LIN {X 0,Y 136.185,Z 195.521,A -85,B 0,C 180,E1 -24638.251,E2 -24638.251} C_VEL
LIN {X 0,Y 136.232,Z 195.509,A -85,B 0,C 180,E1 -24641.969,E2 -24641.969} C_VEL
LIN {X 0,Y 136.486,Z 195.483,A -85,B 0,C 180,E1 -24648.113,E2 -24648.113} C_VEL
LIN {X 0,Y 136.58,Z 195.466,A -85,B 0,C 180,E1 -24651.119,E2 -24651.119} C_VEL
LIN {X 0,Y 137.121,Z 195.397,A -85,B 0,C 180,E1 -24660,E2 -24660} C_VEL
LIN {X 0,Y 136.58,Z 195.467,A -85,B 0,C 180,E1 -24668.88,E2 -24668.88} C_VEL
LIN {X 0,Y 136.479,Z 195.483,A -85,B 0,C 180,E1 -24671.955,E2 -24671.955} C_VEL
LIN {X 0,Y 136.232,Z 195.509,A -85,B 0,C 180,E1 -24678.031,E2 -24678.031} C_VEL
LIN {X 0,Y 136.184,Z 195.521,A -85,B 0,C 180,E1 -24681.747,E2 -24681.747} C_VEL
LIN {X 0,Y 136.081,Z 195.533,A -85,B 0,C 180,E1 -24688.612,E2 -24688.612} C_VEL
LIN {X 0,Y 136.067,Z 195.53,A -85,B 0,C 180,E1 -24694.622,E2 -24694.622} C_VEL
LIN {X 0,Y 136.042,Z 195.539,A -85,B 0,C 180,E1 -24699.212,E2 -24699.212} C_VEL
LIN {X 0,Y 135.998,Z 195.539,A -85,B 0,C 180,E1 -24703.665,E2 -24703.665} C_VEL
LIN {X 0,Y 135.999,Z 195.544,A -85,B 0,C 180,E1 -24707.801,E2 -24707.801} C_VEL
LIN {X 0,Y 136.02,Z 195.536,A -85,B 0,C 180,E1 -24711.688,E2 -24711.688} C_VEL
LIN {X 0,Y 136.079,Z 195.534,A -85,B 0,C 180,E1 -24715.725,E2 -24715.725} C_VEL
LIN {X 0,Y 136.142,Z 195.524,A -85,B 0,C 180,E1 -24722.321,E2 -24722.321} C_VEL
LIN {X 0,Y 136.241,Z 195.509,A -85,B 0,C 180,E1 -24728.838,E2 -24728.838} C_VEL
LIN {X 0,Y 136.275,Z 195.507,A -85,B 0,C 180,E1 -24735.062,E2 -24735.062} C_VEL
LIN {X 0,Y 136.496,Z 195.477,A -85,B 0,C 180,E1 -24738.119,E2 -24738.119} C_VEL
LIN {X 0,Y 136.599,Z 195.469,A -85,B 0,C 180,E1 -24741.126,E2 -24741.126} C_VEL
LIN {X 0,Y 137.127,Z 195.405,A -85,B 0,C 180,E1 -24750.005,E2 -24750.005} C_VEL
LIN {X 0,Y 136.602,Z 195.469,A -85,B 0,C 180,E1 -24758.883,E2 -24758.883} C_VEL
LIN {X 0,Y 136.494,Z 195.477,A -85,B 0,C 180,E1 -24761.959,E2 -24761.959} C_VEL
LIN {X 0,Y 136.243,Z 195.513,A -85,B 0,C 180,E1 -24768.034,E2 -24768.034} C_VEL
LIN {X 0,Y 136.191,Z 195.515,A -85,B 0,C 180,E1 -24771.74,E2 -24771.74} C_VEL
LIN {X 0,Y 136.067,Z 195.533,A -85,B 0,C 180,E1 -24778.59,E2 -24778.59} C_VEL
LIN {X 0,Y 136.046,Z 195.539,A -85,B 0,C 180,E1 -24784.633,E2 -24784.633} C_VEL
LIN {X 0,Y 136.03,Z 195.536,A -85,B 0,C 180,E1 -24789.198,E2 -24789.198} C_VEL
LIN {X 0,Y 135.985,Z 195.545,A -85,B 0,C 180,E1 -24793.652,E2 -24793.652} C_VEL
LIN {X 0,Y 136.055,Z 195.531,A -85,B 0,C 180,E1 -24797.815,E2 -24797.815} C_VEL
LIN {X 0,Y 136.646,Z 195.462,A -85,B 0,C 180,E1 -24805.546,E2 -24805.546} C_VEL
LIN {X 0,Y 136.746,Z 195.503,A -85,B 0,C 180,E1 -24807.341,E2 -24807.341} C_VEL
LIN {X 0,Y 136.371,Z 198.151,A -85,B 0,C 180,E1 -24810.347,E2 -24810.347} C_VEL
LIN {X 0,Y 135.106,Z 204.061,A -85,B 0,C 180,E1 -24817.037,E2 -24817.037} C_VEL
LIN {X 0,Y 134.337,Z 209.498,A -85,B 0,C 180,E1 -24823.278,E2 -24823.278} C_VEL
LIN {X 0,Y 135.028,Z 216.694,A -85,B 0,C 180,E1 -24831.49,E2 -24831.49} C_VEL
LIN {X 0,Y 135.742,Z 218.107,A -85,B 0,C 180,E1 -24833.047,E2 -24833.047} C_VEL
LIN {X 0,Y 136.988,Z 230.698,A -85,B 0,C 180,E1 -24835.218,E2 -24835.218} C_VEL
LIN {X 0,Y 137.062,Z 238.583,A -85,B 0,C 180,E1 -24837.061,E2 -24837.061} C_VEL
LIN {X 0,Y 136.922,Z 249.84,A -85,B 0,C 180,E1 -24840.368,E2 -24840.368} C_VEL
LIN {X 0,Y 136.724,Z 258.747,A -85,B 0,C 180,E1 -24843.684,E2 -24843.684} C_VEL
LIN {X 0,Y 137.067,Z 268.382,A -85,B 0,C 180,E1 -24848.106,E2 -24848.106} C_VEL
LIN {X 0,Y 138.376,Z 276.216,A -85,B 0,C 180,E1 -24852.466,E2 -24852.466} C_VEL
LIN {X 0,Y 140.855,Z 283.522,A -85,B 0,C 180,E1 -24857.42,E2 -24857.42} C_VEL
LIN {X 0,Y 144.239,Z 288.609,A -85,B 0,C 180,E1 -24861.435,E2 -24861.435} C_VEL
LIN {X 0,Y 150.239,Z 293.791,A -85,B 0,C 180,E1 -24866.385,E2 -24866.385} C_VEL
LIN {X 0,Y 155.761,Z 296.577,A -85,B 0,C 180,E1 -24869.757,E2 -24869.757} C_VEL
LIN {X 0,Y 164.409,Z 298.876,A -85,B 0,C 180,E1 -24873.76,E2 -24873.76} C_VEL
LIN {X 0,Y 169.182,Z 299.414,A -85,B 0,C 180,E1 -24875.562,E2 -24875.562} C_VEL
LIN {X 0,Y 173.9,Z 299.584,A -85,B 0,C 180,E1 -24877.316,E2 -24877.316} C_VEL
LIN {X 0,Y 177.161,Z 299.686,A -85,B 0,C 180,E1 -24879.4,E2 -24879.4} C_VEL
LIN {X 0,Y 179.785,Z 299.794,A -85,B 0,C 180,E1 -24881.648,E2 -24881.648} C_VEL
LIN {X 0,Y 180.759,Z 300.28,A -85,B 0,C 180,E1 -24884.415,E2 -24884.415} C_VEL
LIN {X 0,Y 179.098,Z 300.692,A -85,B 0,C 180,E1 -24885.058,E2 -24885.058} C_VEL
LIN {X 0,Y 169.032,Z 302.328,A -85,B 0,C 180,E1 -24888.294,E2 -24888.294} C_VEL
LIN {X 0,Y 159.982,Z 302.764,A -85,B 0,C 180,E1 -24892.042,E2 -24892.042} C_VEL
LIN {X 0,Y 152.204,Z 302.126,A -85,B 0,C 180,E1 -24896.347,E2 -24896.347} C_VEL
LIN {X 0,Y 146.052,Z 300.499,A -85,B 0,C 180,E1 -24901.232,E2 -24901.232} C_VEL
LIN {X 0,Y 141.369,Z 297.748,A -85,B 0,C 180,E1 -24906.56,E2 -24906.56} C_VEL
LIN {X 0,Y 138.541,Z 293.901,A -85,B 0,C 180,E1 -24912.275,E2 -24912.275} C_VEL
LIN {X 0,Y 137.647,Z 288.888,A -85,B 0,C 180,E1 -24918.211,E2 -24918.211} C_VEL
LIN {X 0,Y 138.129,Z 284.139,A -85,B 0,C 180,E1 -24922.688,E2 -24922.688} C_VEL
LIN {X 0,Y 139.011,Z 279.298,A -85,B 0,C 180,E1 -24926.372,E2 -24926.372} C_VEL
LIN {X 0,Y 139.186,Z 274.258,A -85,B 0,C 180,E1 -24929.272,E2 -24929.272} C_VEL
LIN {X 0,Y 138.948,Z 267.938,A -85,B 0,C 180,E1 -24932.169,E2 -24932.169} C_VEL
LIN {X 0,Y 138.845,Z 258.138,A -85,B 0,C 180,E1 -24935.806,E2 -24935.806} C_VEL
LIN {X 0,Y 138.881,Z 248.296,A -85,B 0,C 180,E1 -24938.727,E2 -24938.727} C_VEL
LIN {X 0,Y 138.845,Z 240.573,A -85,B 0,C 180,E1 -24940.568,E2 -24940.568} C_VEL
LIN {X 0,Y 137.226,Z 227.363,A -85,B 0,C 180,E1 -24942.797,E2 -24942.797} C_VEL
LIN {X 0,Y 136.724,Z 219.646,A -85,B 0,C 180,E1 -24943.863,E2 -24943.863} C_VEL
LIN {X 0,Y 135.578,Z 215.399,A -85,B 0,C 180,E1 -24948.116,E2 -24948.116} C_VEL
LIN {X 0,Y 137.903,Z 204.848,A -85,B 0,C 180,E1 -24958.841,E2 -24958.841} C_VEL
LIN {X 0,Y 138.417,Z 203.162,A -85,B 0,C 180,E1 -24960.508,E2 -24960.508} C_VEL
LIN {X 0,Y 136.935,Z 197.26,A -85,B 0,C 180,E1 -24966.418,E2 -24966.418} C_VEL
LIN {X 0,Y 136.522,Z 195.476,A -85,B 0,C 180,E1 -24968.441,E2 -24968.441} C_VEL
LIN {X 0,Y 136.062,Z 195.532,A -85,B 0,C 180,E1 -24976.307,E2 -24976.307} C_VEL
LIN {X 0,Y 136.08,Z 195.534,A -85,B 0,C 180,E1 -24981.702,E2 -24981.702} C_VEL
LIN {X 0,Y 136.082,Z 195.528,A -85,B 0,C 180,E1 -24985.714,E2 -24985.714} C_VEL
LIN {X 0,Y 136.072,Z 195.533,A -85,B 0,C 180,E1 -24991.108,E2 -24991.108} C_VEL
LIN {X 0,Y 135.507,Z 195.614,A -85,B 0,C 180,E1 -24993.578,E2 -24993.578} C_VEL
LIN {X 0,Y 133.984,Z 195.811,A -85,B 0,C 180,E1 -24996.016,E2 -24996.016} C_VEL
LIN {X 0,Y 129.487,Z 196.359,A -85,B 0,C 180,E1 -25002.741,E2 -25002.741} C_VEL
LIN {X 0,Y 129.187,Z 196.388,A -85,B 0,C 180,E1 -25004.52,E2 -25004.52} C_VEL
LIN {X 0,Y 129.405,Z 196.365,A -85,B 0,C 180,E1 -25007.819,E2 -25007.819} C_VEL
LIN {X 0,Y 129.506,Z 196.349,A -85,B 0,C 180,E1 -25010.63,E2 -25010.63} C_VEL
LIN {X 0,Y 130.077,Z 196.274,A -85,B 0,C 180,E1 -25020,E2 -25020} C_VEL
LIN {X 0,Y 129.505,Z 196.349,A -85,B 0,C 180,E1 -25029.369,E2 -25029.369} C_VEL
LIN {X 0,Y 129.381,Z 196.37,A -85,B 0,C 180,E1 -25032.549,E2 -25032.549} C_VEL
LIN {X 0,Y 129.142,Z 196.396,A -85,B 0,C 180,E1 -25039.058,E2 -25039.058} C_VEL
LIN {X 0,Y 129.096,Z 196.404,A -85,B 0,C 180,E1 -25042.4,E2 -25042.4} C_VEL
LIN {X 0,Y 129.006,Z 196.415,A -85,B 0,C 180,E1 -25049.36,E2 -25049.36} C_VEL
LIN {X 0,Y 128.981,Z 196.413,A -85,B 0,C 180,E1 -25055.191,E2 -25055.191} C_VEL
LIN {X 0,Y 128.944,Z 196.421,A -85,B 0,C 180,E1 -25060.848,E2 -25060.848} C_VEL
LIN {X 0,Y 128.917,Z 196.424,A -85,B 0,C 180,E1 -25065.13,E2 -25065.13} C_VEL
LIN {X 0,Y 128.935,Z 196.42,A -85,B 0,C 180,E1 -25069.739,E2 -25069.739} C_VEL
LIN {X 0,Y 128.974,Z 196.419,A -85,B 0,C 180,E1 -25074.822,E2 -25074.822} C_VEL
LIN {X 0,Y 129.046,Z 196.404,A -85,B 0,C 180,E1 -25080.655,E2 -25080.655} C_VEL
LIN {X 0,Y 129.104,Z 196.398,A -85,B 0,C 180,E1 -25087.732,E2 -25087.732} C_VEL
LIN {X 0,Y 129.155,Z 196.396,A -85,B 0,C 180,E1 -25090.949,E2 -25090.949} C_VEL
LIN {X 0,Y 129.415,Z 196.358,A -85,B 0,C 180,E1 -25097.824,E2 -25097.824} C_VEL
LIN {X 0,Y 129.523,Z 196.351,A -85,B 0,C 180,E1 -25100.637,E2 -25100.637} C_VEL
LIN {X 0,Y 130.084,Z 196.282,A -85,B 0,C 180,E1 -25110.005,E2 -25110.005} C_VEL
LIN {X 0,Y 129.526,Z 196.351,A -85,B 0,C 180,E1 -25119.373,E2 -25119.373} C_VEL
LIN {X 0,Y 129.396,Z 196.36,A -85,B 0,C 180,E1 -25122.553,E2 -25122.553} C_VEL
LIN {X 0,Y 129.153,Z 196.396,A -85,B 0,C 180,E1 -25129.061,E2 -25129.061} C_VEL
LIN {X 0,Y 129.083,Z 196.4,A -85,B 0,C 180,E1 -25132.408,E2 -25132.408} C_VEL
LIN {X 0,Y 129.004,Z 196.409,A -85,B 0,C 180,E1 -25139.366,E2 -25139.366} C_VEL
LIN {X 0,Y 128.962,Z 196.42,A -85,B 0,C 180,E1 -25145.17,E2 -25145.17} C_VEL
LIN {X 0,Y 128.929,Z 196.424,A -85,B 0,C 180,E1 -25150.86,E2 -25150.86} C_VEL
LIN {X 0,Y 128.926,Z 196.422,A -85,B 0,C 180,E1 -25155.132,E2 -25155.132} C_VEL
LIN {X 0,Y 129.068,Z 196.406,A -85,B 0,C 180,E1 -25159.677,E2 -25159.677} C_VEL
LIN {X 0,Y 129.697,Z 196.328,A -85,B 0,C 180,E1 -25167.189,E2 -25167.189} C_VEL
LIN {X 0,Y 129.606,Z 196.58,A -85,B 0,C 180,E1 -25168.174,E2 -25168.174} C_VEL
LIN {X 0,Y 128.824,Z 200.1,A -85,B 0,C 180,E1 -25172.373,E2 -25172.373} C_VEL
LIN {X 0,Y 127.675,Z 205.925,A -85,B 0,C 180,E1 -25179.367,E2 -25179.367} C_VEL
LIN {X 0,Y 127.901,Z 216.003,A -85,B 0,C 180,E1 -25191.553,E2 -25191.553} C_VEL
LIN {X 0,Y 129.041,Z 218.151,A -85,B 0,C 180,E1 -25194.041,E2 -25194.041} C_VEL
LIN {X 0,Y 130.451,Z 231.526,A -85,B 0,C 180,E1 -25196.525,E2 -25196.525} C_VEL
LIN {X 0,Y 130.298,Z 241.723,A -85,B 0,C 180,E1 -25199.228,E2 -25199.228} C_VEL
LIN {X 0,Y 130.316,Z 250.105,A -85,B 0,C 180,E1 -25201.932,E2 -25201.932} C_VEL
LIN {X 0,Y 130.224,Z 260.548,A -85,B 0,C 180,E1 -25206.197,E2 -25206.197} C_VEL
LIN {X 0,Y 131.035,Z 269.788,A -85,B 0,C 180,E1 -25210.82,E2 -25210.82} C_VEL
LIN {X 0,Y 132.753,Z 277.34,A -85,B 0,C 180,E1 -25215.35,E2 -25215.35} C_VEL
LIN {X 0,Y 135.392,Z 283.506,A -85,B 0,C 180,E1 -25219.719,E2 -25219.719} C_VEL
LIN {X 0,Y 139.207,Z 288.632,A -85,B 0,C 180,E1 -25223.822,E2 -25223.822} C_VEL
LIN {X 0,Y 143.978,Z 292.767,A -85,B 0,C 180,E1 -25227.628,E2 -25227.628} C_VEL
LIN {X 0,Y 149.639,Z 295.964,A -85,B 0,C 180,E1 -25231.107,E2 -25231.107} C_VEL
LIN {X 0,Y 158.53,Z 298.838,A -85,B 0,C 180,E1 -25235.192,E2 -25235.192} C_VEL
LIN {X 0,Y 163.424,Z 299.685,A -85,B 0,C 180,E1 -25237.018,E2 -25237.018} C_VEL
LIN {X 0,Y 168.224,Z 300.154,A -85,B 0,C 180,E1 -25238.805,E2 -25238.805} C_VEL
LIN {X 0,Y 171.426,Z 300.516,A -85,B 0,C 180,E1 -25240.992,E2 -25240.992} C_VEL
LIN {X 0,Y 173.235,Z 300.876,A -85,B 0,C 180,E1 -25243.089,E2 -25243.089} C_VEL
LIN {X 0,Y 173.376,Z 300.975,A -85,B 0,C 180,E1 -25243.56,E2 -25243.56} C_VEL
LIN {X 0,Y 163.826,Z 301.929,A -85,B 0,C 180,E1 -25246.651,E2 -25246.651} C_VEL
LIN {X 0,Y 154.492,Z 301.857,A -85,B 0,C 180,E1 -25250.436,E2 -25250.436} C_VEL
LIN {X 0,Y 146.459,Z 300.764,A -85,B 0,C 180,E1 -25254.837,E2 -25254.837} C_VEL
LIN {X 0,Y 140.058,Z 298.71,A -85,B 0,C 180,E1 -25259.877,E2 -25259.877} C_VEL
LIN {X 0,Y 135.211,Z 295.569,A -85,B 0,C 180,E1 -25265.424,E2 -25265.424} C_VEL
LIN {X 0,Y 132.259,Z 291.351,A -85,B 0,C 180,E1 -25271.403,E2 -25271.403} C_VEL
LIN {X 0,Y 131.335,Z 285.974,A -85,B 0,C 180,E1 -25277.636,E2 -25277.636} C_VEL
LIN {X 0,Y 132.172,Z 278.979,A -85,B 0,C 180,E1 -25283.89,E2 -25283.89} C_VEL
LIN {X 0,Y 132.823,Z 274.537,A -85,B 0,C 180,E1 -25286.962,E2 -25286.962} C_VEL
LIN {X 0,Y 132.739,Z 268.673,A -85,B 0,C 180,E1 -25289.995,E2 -25289.995} C_VEL
LIN {X 0,Y 132.359,Z 258.286,A -85,B 0,C 180,E1 -25294.182,E2 -25294.182} C_VEL
LIN {X 0,Y 132.311,Z 248.78,A -85,B 0,C 180,E1 -25297.242,E2 -25297.242} C_VEL
LIN {X 0,Y 132.387,Z 241.482,A -85,B 0,C 180,E1 -25299.159,E2 -25299.159} C_VEL
LIN {X 0,Y 130.94,Z 230.536,A -85,B 0,C 180,E1 -25301.214,E2 -25301.214} C_VEL
LIN {X 0,Y 130.002,Z 219.592,A -85,B 0,C 180,E1 -25302.881,E2 -25302.881} C_VEL
LIN {X 0,Y 128.571,Z 215.257,A -85,B 0,C 180,E1 -25307.491,E2 -25307.491} C_VEL
LIN {X 0,Y 130.761,Z 204.687,A -85,B 0,C 180,E1 -25318.923,E2 -25318.923} C_VEL
LIN {X 0,Y 131.142,Z 202.729,A -85,B 0,C 180,E1 -25320.968,E2 -25320.968} C_VEL
LIN {X 0,Y 129.529,Z 196.349,A -85,B 0,C 180,E1 -25327.858,E2 -25327.858} C_VEL
LIN {X 0,Y 129.012,Z 196.412,A -85,B 0,C 180,E1 -25335.08,E2 -25335.08} C_VEL
LIN {X 0,Y 129.001,Z 196.414,A -85,B 0,C 180,E1 -25339.696,E2 -25339.696} C_VEL
LIN {X 0,Y 129.014,Z 196.409,A -85,B 0,C 180,E1 -25344.788,E2 -25344.788} C_VEL
LIN {X 0,Y 128.983,Z 196.414,A -85,B 0,C 180,E1 -25351.041,E2 -25351.041} C_VEL
LIN {X 0,Y 129.096,Z 196.404,A -85,B 0,C 180,E1 -25357.726,E2 -25357.726} C_VEL
LIN {X 0,Y 129.143,Z 196.396,A -85,B 0,C 180,E1 -25360.942,E2 -25360.942} C_VEL
LIN {X 0,Y 129.187,Z 196.388,A -85,B 0,C 180,E1 -25364.52,E2 -25364.52} C_VEL
LIN {X 0,Y 128.54,Z 196.474,A -85,B 0,C 180,E1 -25367.126,E2 -25367.126} C_VEL
LIN {X 0,Y 126.996,Z 196.662,A -85,B 0,C 180,E1 -25369.701,E2 -25369.701} C_VEL
LIN {X 0,Y 123.522,Z 197.098,A -85,B 0,C 180,E1 -25374.983,E2 -25374.983} C_VEL
LIN {X 0,Y 122.765,Z 197.19,A -85,B 0,C 180,E1 -25377.761,E2 -25377.761} C_VEL
LIN {X 0,Y 122.81,Z 197.176,A -85,B 0,C 180,E1 -25378.697,E2 -25378.697} C_VEL
LIN {X 0,Y 123.03,Z 197.152,A -85,B 0,C 180,E1 -25380,E2 -25380} C_VEL
LIN {X 0,Y 122.404,Z 197.231,A -85,B 0,C 180,E1 -25387.183,E2 -25387.183} C_VEL
LIN {X 0,Y 122.352,Z 197.245,A -85,B 0,C 180,E1 -25392.474,E2 -25392.474} C_VEL
LIN {X 0,Y 122.034,Z 197.283,A -85,B 0,C 180,E1 -25400.215,E2 -25400.215} C_VEL
LIN {X 0,Y 121.97,Z 197.29,A -85,B 0,C 180,E1 -25403.787,E2 -25403.787} C_VEL
LIN {X 0,Y 121.918,Z 197.299,A -85,B 0,C 180,E1 -25410.166,E2 -25410.166} C_VEL
LIN {X 0,Y 121.902,Z 197.298,A -85,B 0,C 180,E1 -25416.192,E2 -25416.192} C_VEL
LIN {X 0,Y 121.877,Z 197.299,A -85,B 0,C 180,E1 -25421.45,E2 -25421.45} C_VEL
LIN {X 0,Y 121.865,Z 197.304,A -85,B 0,C 180,E1 -25428.565,E2 -25428.565} C_VEL
LIN {X 0,Y 121.926,Z 197.297,A -85,B 0,C 180,E1 -25434.808,E2 -25434.808} C_VEL
LIN {X 0,Y 121.936,Z 197.288,A -85,B 0,C 180,E1 -25439.831,E2 -25439.831} C_VEL
LIN {X 0,Y 121.98,Z 197.29,A -85,B 0,C 180,E1 -25446.221,E2 -25446.221} C_VEL
LIN {X 0,Y 122.044,Z 197.278,A -85,B 0,C 180,E1 -25449.793,E2 -25449.793} C_VEL
LIN {X 0,Y 122.362,Z 197.236,A -85,B 0,C 180,E1 -25457.531,E2 -25457.531} C_VEL
LIN {X 0,Y 122.45,Z 197.231,A -85,B 0,C 180,E1 -25460.091,E2 -25460.091} C_VEL
LIN {X 0,Y 122.61,Z 197.208,A -85,B 0,C 180,E1 -25466.719,E2 -25466.719} C_VEL
LIN {X 0,Y 123.039,Z 197.16,A -85,B 0,C 180,E1 -25470.005,E2 -25470.005} C_VEL
LIN {X 0,Y 122.453,Z 197.23,A -85,B 0,C 180,E1 -25476.596,E2 -25476.596} C_VEL
LIN {X 0,Y 122.454,Z 197.231,A -85,B 0,C 180,E1 -25479.92,E2 -25479.92} C_VEL
LIN {X 0,Y 122.264,Z 197.248,A -85,B 0,C 180,E1 -25483.298,E2 -25483.298} C_VEL
LIN {X 0,Y 122.045,Z 197.278,A -85,B 0,C 180,E1 -25490.218,E2 -25490.218} C_VEL
LIN {X 0,Y 121.954,Z 197.293,A -85,B 0,C 180,E1 -25493.796,E2 -25493.796} C_VEL
LIN {X 0,Y 121.92,Z 197.29,A -85,B 0,C 180,E1 -25500.156,E2 -25500.156} C_VEL
LIN {X 0,Y 121.886,Z 197.301,A -85,B 0,C 180,E1 -25506.173,E2 -25506.173} C_VEL
LIN {X 0,Y 121.87,Z 197.303,A -85,B 0,C 180,E1 -25511.437,E2 -25511.437} C_VEL
LIN {X 0,Y 121.954,Z 197.29,A -85,B 0,C 180,E1 -25518.525,E2 -25518.525} C_VEL
LIN {X 0,Y 122.392,Z 197.237,A -85,B 0,C 180,E1 -25524.955,E2 -25524.955} C_VEL
LIN {X 0,Y 122.572,Z 197.217,A -85,B 0,C 180,E1 -25527.97,E2 -25527.97} C_VEL
LIN {X 0,Y 122.43,Z 197.446,A -85,B 0,C 180,E1 -25528.893,E2 -25528.893} C_VEL
LIN {X 0,Y 121.041,Z 203.093,A -85,B 0,C 180,E1 -25536.019,E2 -25536.019} C_VEL
LIN {X 0,Y 120.198,Z 208.532,A -85,B 0,C 180,E1 -25543.002,E2 -25543.002} C_VEL
LIN {X 0,Y 121.419,Z 216.63,A -85,B 0,C 180,E1 -25553.353,E2 -25553.353} C_VEL
LIN {X 0,Y 122.455,Z 218.222,A -85,B 0,C 180,E1 -25555.268,E2 -25555.268} C_VEL
LIN {X 0,Y 123.811,Z 230.309,A -85,B 0,C 180,E1 -25557.56,E2 -25557.56} C_VEL
LIN {X 0,Y 123.78,Z 239.315,A -85,B 0,C 180,E1 -25560,E2 -25560} C_VEL
LIN {X 0,Y 123.839,Z 247.995,A -85,B 0,C 180,E1 -25562.847,E2 -25562.847} C_VEL
LIN {X 0,Y 123.816,Z 256.984,A -85,B 0,C 180,E1 -25566.519,E2 -25566.519} C_VEL
LIN {X 0,Y 124.553,Z 266.798,A -85,B 0,C 180,E1 -25571.391,E2 -25571.391} C_VEL
LIN {X 0,Y 126.295,Z 274.829,A -85,B 0,C 180,E1 -25576.155,E2 -25576.155} C_VEL
LIN {X 0,Y 128.991,Z 281.428,A -85,B 0,C 180,E1 -25580.742,E2 -25580.742} C_VEL
LIN {X 0,Y 132.887,Z 286.953,A -85,B 0,C 180,E1 -25585.031,E2 -25585.031} C_VEL
LIN {X 0,Y 137.827,Z 291.501,A -85,B 0,C 180,E1 -25588.975,E2 -25588.975} C_VEL
LIN {X 0,Y 143.645,Z 295.113,A -85,B 0,C 180,E1 -25592.561,E2 -25592.561} C_VEL
LIN {X 0,Y 152.763,Z 298.551,A -85,B 0,C 180,E1 -25596.733,E2 -25596.733} C_VEL
LIN {X 0,Y 157.766,Z 299.707,A -85,B 0,C 180,E1 -25598.584,E2 -25598.584} C_VEL
LIN {X 0,Y 162.602,Z 300.471,A -85,B 0,C 180,E1 -25600.416,E2 -25600.416} C_VEL
LIN {X 0,Y 164.231,Z 300.782,A -85,B 0,C 180,E1 -25601.506,E2 -25601.506} C_VEL
LIN {X 0,Y 165.279,Z 301.096,A -85,B 0,C 180,E1 -25602.817,E2 -25602.817} C_VEL
LIN {X 0,Y 153.825,Z 301.115,A -85,B 0,C 180,E1 -25606.734,E2 -25606.734} C_VEL
LIN {X 0,Y 143.683,Z 299.838,A -85,B 0,C 180,E1 -25611.501,E2 -25611.501} C_VEL
LIN {X 0,Y 137.381,Z 298.062,A -85,B 0,C 180,E1 -25615.75,E2 -25615.75} C_VEL
LIN {X 0,Y 131.486,Z 295.075,A -85,B 0,C 180,E1 -25621.241,E2 -25621.241} C_VEL
LIN {X 0,Y 127.372,Z 291.003,A -85,B 0,C 180,E1 -25627.274,E2 -25627.274} C_VEL
LIN {X 0,Y 125.362,Z 285.858,A -85,B 0,C 180,E1 -25633.716,E2 -25633.716} C_VEL
LIN {X 0,Y 125.367,Z 279.352,A -85,B 0,C 180,E1 -25640.313,E2 -25640.313} C_VEL
LIN {X 0,Y 126.463,Z 273.206,A -85,B 0,C 180,E1 -25645.213,E2 -25645.213} C_VEL
LIN {X 0,Y 126.561,Z 269.101,A -85,B 0,C 180,E1 -25647.608,E2 -25647.608} C_VEL
LIN {X 0,Y 126.164,Z 262.216,A -85,B 0,C 180,E1 -25650.793,E2 -25650.793} C_VEL
LIN {X 0,Y 125.883,Z 252.74,A -85,B 0,C 180,E1 -25654.398,E2 -25654.398} C_VEL
LIN {X 0,Y 125.837,Z 243.471,A -85,B 0,C 180,E1 -25657.214,E2 -25657.214} C_VEL
LIN {X 0,Y 125.848,Z 240.423,A -85,B 0,C 180,E1 -25658.02,E2 -25658.02} C_VEL
LIN {X 0,Y 124.113,Z 227.939,A -85,B 0,C 180,E1 -25660.393,E2 -25660.393} C_VEL
LIN {X 0,Y 123.416,Z 219.608,A -85,B 0,C 180,E1 -25661.699,E2 -25661.699} C_VEL
LIN {X 0,Y 121.915,Z 216.583,A -85,B 0,C 180,E1 -25665.029,E2 -25665.029} C_VEL
LIN {X 0,Y 123.597,Z 204.577,A -85,B 0,C 180,E1 -25678.897,E2 -25678.897} C_VEL
LIN {X 0,Y 123.953,Z 202.983,A -85,B 0,C 180,E1 -25680.677,E2 -25680.677} C_VEL
LIN {X 0,Y 122.664,Z 197.671,A -85,B 0,C 180,E1 -25686.665,E2 -25686.665} C_VEL
LIN {X 0,Y 122.522,Z 197.223,A -85,B 0,C 180,E1 -25687.47,E2 -25687.47} C_VEL
LIN {X 0,Y 121.914,Z 197.294,A -85,B 0,C 180,E1 -25696.229,E2 -25696.229} C_VEL
LIN {X 0,Y 121.904,Z 197.3,A -85,B 0,C 180,E1 -25700.641,E2 -25700.641} C_VEL
LIN {X 0,Y 121.966,Z 197.286,A -85,B 0,C 180,E1 -25704.814,E2 -25704.814} C_VEL
LIN {X 0,Y 121.919,Z 197.299,A -85,B 0,C 180,E1 -25709.833,E2 -25709.833} C_VEL
LIN {X 0,Y 121.971,Z 197.29,A -85,B 0,C 180,E1 -25716.212,E2 -25716.212} C_VEL
LIN {X 0,Y 122.034,Z 197.283,A -85,B 0,C 180,E1 -25719.785,E2 -25719.785} C_VEL
LIN {X 0,Y 122.352,Z 197.245,A -85,B 0,C 180,E1 -25727.525,E2 -25727.525} C_VEL
LIN {X 0,Y 122.435,Z 197.229,A -85,B 0,C 180,E1 -25730.084,E2 -25730.084} C_VEL
LIN {X 0,Y 122.81,Z 197.176,A -85,B 0,C 180,E1 -25738.697,E2 -25738.697} C_VEL
LIN {X 0,Y 122.687,Z 197.195,A -85,B 0,C 180,E1 -25740.519,E2 -25740.519} C_VEL
LIN {X 0,Y 121.428,Z 197.36,A -85,B 0,C 180,E1 -25743.221,E2 -25743.221} C_VEL
LIN {X 0,Y 118.021,Z 197.783,A -85,B 0,C 180,E1 -25747.739,E2 -25747.739} C_VEL
LIN {X 0,Y 115.36,Z 198.116,A -85,B 0,C 180,E1 -25752.571,E2 -25752.571} C_VEL
LIN {X 0,Y 115.181,Z 198.137,A -85,B 0,C 180,E1 -25753.579,E2 -25753.579} C_VEL
LIN {X 0,Y 115.001,Z 198.153,A -85,B 0,C 180,E1 -25757.792,E2 -25757.792} C_VEL
LIN {X 0,Y 114.935,Z 198.167,A -85,B 0,C 180,E1 -25763.493,E2 -25763.493} C_VEL
LIN {X 0,Y 114.852,Z 198.178,A -85,B 0,C 180,E1 -25771.065,E2 -25771.065} C_VEL
LIN {X 0,Y 114.793,Z 198.186,A -85,B 0,C 180,E1 -25777.751,E2 -25777.751} C_VEL
LIN {X 0,Y 114.788,Z 198.179,A -85,B 0,C 180,E1 -25782.726,E2 -25782.726} C_VEL
LIN {X 0,Y 114.788,Z 198.186,A -85,B 0,C 180,E1 -25787.672,E2 -25787.672} C_VEL
LIN {X 0,Y 114.791,Z 198.181,A -85,B 0,C 180,E1 -25792.742,E2 -25792.742} C_VEL
LIN {X 0,Y 114.862,Z 198.171,A -85,B 0,C 180,E1 -25798.938,E2 -25798.938} C_VEL
LIN {X 0,Y 114.943,Z 198.165,A -85,B 0,C 180,E1 -25806.513,E2 -25806.513} C_VEL
LIN {X 0,Y 115.012,Z 198.158,A -85,B 0,C 180,E1 -25812.216,E2 -25812.216} C_VEL
LIN {X 0,Y 115.283,Z 198.117,A -85,B 0,C 180,E1 -25817.266,E2 -25817.266} C_VEL
LIN {X 0,Y 115.394,Z 198.109,A -85,B 0,C 180,E1 -25823.009,E2 -25823.009} C_VEL
LIN {X 0,Y 115.992,Z 198.038,A -85,B 0,C 180,E1 -25830.005,E2 -25830.005} C_VEL
LIN {X 0,Y 115.395,Z 198.109,A -85,B 0,C 180,E1 -25837.002,E2 -25837.002} C_VEL
LIN {X 0,Y 115.288,Z 198.117,A -85,B 0,C 180,E1 -25842.745,E2 -25842.745} C_VEL
LIN {X 0,Y 115.013,Z 198.158,A -85,B 0,C 180,E1 -25847.796,E2 -25847.796} C_VEL
LIN {X 0,Y 114.924,Z 198.167,A -85,B 0,C 180,E1 -25853.465,E2 -25853.465} C_VEL
LIN {X 0,Y 114.852,Z 198.173,A -85,B 0,C 180,E1 -25861.054,E2 -25861.054} C_VEL
LIN {X 0,Y 114.78,Z 198.182,A -85,B 0,C 180,E1 -25867.763,E2 -25867.763} C_VEL
LIN {X 0,Y 114.787,Z 198.188,A -85,B 0,C 180,E1 -25872.717,E2 -25872.717} C_VEL
LIN {X 0,Y 114.855,Z 198.171,A -85,B 0,C 180,E1 -25877.694,E2 -25877.694} C_VEL
LIN {X 0,Y 115.104,Z 198.146,A -85,B 0,C 180,E1 -25882.546,E2 -25882.546} C_VEL
LIN {X 0,Y 115.531,Z 198.089,A -85,B 0,C 180,E1 -25886.805,E2 -25886.805} C_VEL
LIN {X 0,Y 115.156,Z 198.209,A -85,B 0,C 180,E1 -25889.606,E2 -25889.606} C_VEL
LIN {X 0,Y 113.632,Z 204.621,A -85,B 0,C 180,E1 -25898.217,E2 -25898.217} C_VEL
LIN {X 0,Y 114.055,Z 215.396,A -85,B 0,C 180,E1 -25912.921,E2 -25912.921} C_VEL
LIN {X 0,Y 115.943,Z 218.292,A -85,B 0,C 180,E1 -25916.634,E2 -25916.634} C_VEL
LIN {X 0,Y 117.345,Z 230.572,A -85,B 0,C 180,E1 -25919.142,E2 -25919.142} C_VEL
LIN {X 0,Y 117.352,Z 240.715,A -85,B 0,C 180,E1 -25922.145,E2 -25922.145} C_VEL
LIN {X 0,Y 117.428,Z 247.889,A -85,B 0,C 180,E1 -25924.721,E2 -25924.721} C_VEL
LIN {X 0,Y 117.544,Z 256.775,A -85,B 0,C 180,E1 -25928.597,E2 -25928.597} C_VEL
LIN {X 0,Y 118.676,Z 266.569,A -85,B 0,C 180,E1 -25933.703,E2 -25933.703} C_VEL
LIN {X 0,Y 120.718,Z 274.52,A -85,B 0,C 180,E1 -25938.675,E2 -25938.675} C_VEL
LIN {X 0,Y 123.873,Z 281.193,A -85,B 0,C 180,E1 -25943.4,E2 -25943.4} C_VEL
LIN {X 0,Y 128.296,Z 286.792,A -85,B 0,C 180,E1 -25947.751,E2 -25947.751} C_VEL
LIN {X 0,Y 133.654,Z 291.404,A -85,B 0,C 180,E1 -25951.725,E2 -25951.725} C_VEL
LIN {X 0,Y 139.996,Z 295.141,A -85,B 0,C 180,E1 -25955.262,E2 -25955.262} C_VEL
LIN {X 0,Y 147.121,Z 298.01,A -85,B 0,C 180,E1 -25958.39,E2 -25958.39} C_VEL
LIN {X 0,Y 155.818,Z 300.258,A -85,B 0,C 180,E1 -25961.577,E2 -25961.577} C_VEL
LIN {X 0,Y 156.171,Z 300.467,A -85,B 0,C 180,E1 -25962.3,E2 -25962.3} C_VEL
LIN {X 0,Y 148.804,Z 299.943,A -85,B 0,C 180,E1 -25964.886,E2 -25964.886} C_VEL
LIN {X 0,Y 139.509,Z 298.406,A -85,B 0,C 180,E1 -25969.083,E2 -25969.083} C_VEL
LIN {X 0,Y 131.815,Z 296.006,A -85,B 0,C 180,E1 -25974.086,E2 -25974.086} C_VEL
LIN {X 0,Y 125.687,Z 292.607,A -85,B 0,C 180,E1 -25979.779,E2 -25979.779} C_VEL
LIN {X 0,Y 121.398,Z 288.169,A -85,B 0,C 180,E1 -25986.088,E2 -25986.088} C_VEL
LIN {X 0,Y 119.293,Z 282.668,A -85,B 0,C 180,E1 -25992.863,E2 -25992.863} C_VEL
LIN {X 0,Y 119.127,Z 277.634,A -85,B 0,C 180,E1 -25998.078,E2 -25998.078} C_VEL
LIN {X 0,Y 120.182,Z 270.926,A -85,B 0,C 180,E1 -26003.79,E2 -26003.79} C_VEL
LIN {X 0,Y 120.434,Z 267.784,A -85,B 0,C 180,E1 -26005.811,E2 -26005.811} C_VEL
LIN {X 0,Y 120.164,Z 262.875,A -85,B 0,C 180,E1 -26008.319,E2 -26008.319} C_VEL
LIN {X 0,Y 119.675,Z 253.186,A -85,B 0,C 180,E1 -26012.339,E2 -26012.339} C_VEL
LIN {X 0,Y 119.44,Z 243.68,A -85,B 0,C 180,E1 -26015.481,E2 -26015.481} C_VEL
LIN {X 0,Y 119.224,Z 238.106,A -85,B 0,C 180,E1 -26016.978,E2 -26016.978} C_VEL
LIN {X 0,Y 117.492,Z 226.356,A -85,B 0,C 180,E1 -26019.245,E2 -26019.245} C_VEL
LIN {X 0,Y 116.824,Z 219.529,A -85,B 0,C 180,E1 -26020.392,E2 -26020.392} C_VEL
LIN {X 0,Y 115.058,Z 216.347,A -85,B 0,C 180,E1 -26024.136,E2 -26024.136} C_VEL
LIN {X 0,Y 114.645,Z 210.351,A -85,B 0,C 180,E1 -26031.575,E2 -26031.575} C_VEL
LIN {X 0,Y 116.424,Z 204.423,A -85,B 0,C 180,E1 -26038.87,E2 -26038.87} C_VEL
LIN {X 0,Y 116.801,Z 203.058,A -85,B 0,C 180,E1 -26040.506,E2 -26040.506} C_VEL
LIN {X 0,Y 115.84,Z 199.143,A -85,B 0,C 180,E1 -26045.188,E2 -26045.188} C_VEL
LIN {X 0,Y 115.587,Z 198.09,A -85,B 0,C 180,E1 -26046.621,E2 -26046.621} C_VEL
LIN {X 0,Y 114.938,Z 198.168,A -85,B 0,C 180,E1 -26052.798,E2 -26052.798} C_VEL
LIN {X 0,Y 114.856,Z 198.171,A -85,B 0,C 180,E1 -26057.694,E2 -26057.694} C_VEL
LIN {X 0,Y 114.846,Z 198.178,A -85,B 0,C 180,E1 -26062.696,E2 -26062.696} C_VEL
LIN {X 0,Y 114.854,Z 198.177,A -85,B 0,C 180,E1 -26068.933,E2 -26068.933} C_VEL
LIN {X 0,Y 114.936,Z 198.166,A -85,B 0,C 180,E1 -26076.505,E2 -26076.505} C_VEL
LIN {X 0,Y 115.002,Z 198.153,A -85,B 0,C 180,E1 -26082.208,E2 -26082.208} C_VEL
LIN {X 0,Y 115.273,Z 198.127,A -85,B 0,C 180,E1 -26087.261,E2 -26087.261} C_VEL
LIN {X 0,Y 115.378,Z 198.109,A -85,B 0,C 180,E1 -26093.002,E2 -26093.002} C_VEL
LIN {X 0,Y 115.982,Z 198.029,A -85,B 0,C 180,E1 -26100,E2 -26100} C_VEL
LIN {X 0,Y 115.37,Z 198.109,A -85,B 0,C 180,E1 -26107.075,E2 -26107.075} C_VEL
LIN {X 0,Y 115.273,Z 198.127,A -85,B 0,C 180,E1 -26112.739,E2 -26112.739} C_VEL
LIN {X 0,Y 115.181,Z 198.137,A -85,B 0,C 180,E1 -26113.579,E2 -26113.579} C_VEL
LIN {X 0,Y 114.289,Z 198.249,A -85,B 0,C 180,E1 -26116.494,E2 -26116.494} C_VEL
LIN {X 0,Y 112.572,Z 198.464,A -85,B 0,C 180,E1 -26119.372,E2 -26119.372} C_VEL
LIN {X 0,Y 107.97,Z 199.032,A -85,B 0,C 180,E1 -26127.392,E2 -26127.392} C_VEL
LIN {X 0,Y 107.694,Z 199.059,A -85,B 0,C 180,E1 -26129.525,E2 -26129.525} C_VEL
LIN {X 0,Y 107.779,Z 199.057,A -85,B 0,C 180,E1 -26132.05,E2 -26132.05} C_VEL
LIN {X 0,Y 107.699,Z 199.069,A -85,B 0,C 180,E1 -26138.468,E2 -26138.468} C_VEL
LIN {X 0,Y 107.672,Z 199.073,A -85,B 0,C 180,E1 -26145.889,E2 -26145.889} C_VEL
LIN {X 0,Y 107.687,Z 199.064,A -85,B 0,C 180,E1 -26151.55,E2 -26151.55} C_VEL
LIN {X 0,Y 107.799,Z 199.053,A -85,B 0,C 180,E1 -26158.57,E2 -26158.57} C_VEL
LIN {X 0,Y 107.907,Z 199.039,A -85,B 0,C 180,E1 -26167.004,E2 -26167.004} C_VEL
LIN {X 0,Y 108.036,Z 199.025,A -85,B 0,C 180,E1 -26174.924,E2 -26174.924} C_VEL
LIN {X 0,Y 108.302,Z 198.991,A -85,B 0,C 180,E1 -26178.78,E2 -26178.78} C_VEL
LIN {X 0,Y 108.461,Z 198.968,A -85,B 0,C 180,E1 -26186.291,E2 -26186.291} C_VEL
LIN {X 0,Y 108.943,Z 198.916,A -85,B 0,C 180,E1 -26190.006,E2 -26190.006} C_VEL
LIN {X 0,Y 108.338,Z 198.989,A -85,B 0,C 180,E1 -26197.461,E2 -26197.461} C_VEL
LIN {X 0,Y 108.205,Z 198.999,A -85,B 0,C 180,E1 -26203.028,E2 -26203.028} C_VEL
LIN {X 0,Y 107.903,Z 199.043,A -85,B 0,C 180,E1 -26209.012,E2 -26209.012} C_VEL
LIN {X 0,Y 107.828,Z 199.052,A -85,B 0,C 180,E1 -26214.149,E2 -26214.149} C_VEL
LIN {X 0,Y 107.778,Z 199.057,A -85,B 0,C 180,E1 -26222.037,E2 -26222.037} C_VEL
LIN {X 0,Y 107.689,Z 199.064,A -85,B 0,C 180,E1 -26228.451,E2 -26228.451} C_VEL
LIN {X 0,Y 107.71,Z 199.064,A -85,B 0,C 180,E1 -26235.876,E2 -26235.876} C_VEL
LIN {X 0,Y 107.926,Z 199.041,A -85,B 0,C 180,E1 -26241.4,E2 -26241.4} C_VEL
LIN {X 0,Y 108.445,Z 198.975,A -85,B 0,C 180,E1 -26247.414,E2 -26247.414} C_VEL
LIN {X 0,Y 107.773,Z 199.152,A -85,B 0,C 180,E1 -26250.72,E2 -26250.72} C_VEL
LIN {X 0,Y 106.414,Z 204.919,A -85,B 0,C 180,E1 -26258.998,E2 -26258.998} C_VEL
LIN {X 0,Y 107.408,Z 215.465,A -85,B 0,C 180,E1 -26274.368,E2 -26274.368} C_VEL
LIN {X 0,Y 109.576,Z 218.376,A -85,B 0,C 180,E1 -26278.277,E2 -26278.277} C_VEL
LIN {X 0,Y 110.926,Z 228.888,A -85,B 0,C 180,E1 -26280.454,E2 -26280.454} C_VEL
LIN {X 0,Y 111.055,Z 239.335,A -85,B 0,C 180,E1 -26283.629,E2 -26283.629} C_VEL
LIN {X 0,Y 111.177,Z 246.549,A -85,B 0,C 180,E1 -26286.352,E2 -26286.352} C_VEL
LIN {X 0,Y 111.536,Z 256.422,A -85,B 0,C 180,E1 -26290.897,E2 -26290.897} C_VEL
LIN {X 0,Y 113.026,Z 266.165,A -85,B 0,C 180,E1 -26296.249,E2 -26296.249} C_VEL
LIN {X 0,Y 115.405,Z 274.093,A -85,B 0,C 180,E1 -26301.432,E2 -26301.432} C_VEL
LIN {X 0,Y 119.836,Z 281.85,A -85,B 0,C 180,E1 -26307.034,E2 -26307.034} C_VEL
LIN {X 0,Y 125.879,Z 288.198,A -85,B 0,C 180,E1 -26312.033,E2 -26312.033} C_VEL
LIN {X 0,Y 132.013,Z 292.623,A -85,B 0,C 180,E1 -26315.847,E2 -26315.847} C_VEL
LIN {X 0,Y 141.618,Z 297.208,A -85,B 0,C 180,E1 -26320.177,E2 -26320.177} C_VEL
LIN {X 0,Y 145.356,Z 298.482,A -85,B 0,C 180,E1 -26321.544,E2 -26321.544} C_VEL
LIN {X 0,Y 143.996,Z 298.507,A -85,B 0,C 180,E1 -26322.931,E2 -26322.931} C_VEL
LIN {X 0,Y 134.421,Z 296.512,A -85,B 0,C 180,E1 -26327.175,E2 -26327.175} C_VEL
LIN {X 0,Y 126.441,Z 293.682,A -85,B 0,C 180,E1 -26332.302,E2 -26332.302} C_VEL
LIN {X 0,Y 120.067,Z 289.899,A -85,B 0,C 180,E1 -26338.204,E2 -26338.204} C_VEL
LIN {X 0,Y 115.581,Z 285.103,A -85,B 0,C 180,E1 -26344.803,E2 -26344.803} C_VEL
LIN {X 0,Y 113.388,Z 279.224,A -85,B 0,C 180,E1 -26351.941,E2 -26351.941} C_VEL
LIN {X 0,Y 113.231,Z 273.897,A -85,B 0,C 180,E1 -26357.448,E2 -26357.448} C_VEL
LIN {X 0,Y 114.204,Z 267.508,A -85,B 0,C 180,E1 -26362.925,E2 -26362.925} C_VEL
LIN {X 0,Y 114.417,Z 265.001,A -85,B 0,C 180,E1 -26364.594,E2 -26364.594} C_VEL
LIN {X 0,Y 113.85,Z 257.708,A -85,B 0,C 180,E1 -26368.226,E2 -26368.226} C_VEL
LIN {X 0,Y 113.439,Z 249.75,A -85,B 0,C 180,E1 -26371.459,E2 -26371.459} C_VEL
LIN {X 0,Y 113.089,Z 239.146,A -85,B 0,C 180,E1 -26374.93,E2 -26374.93} C_VEL
LIN {X 0,Y 111.837,Z 230.868,A -85,B 0,C 180,E1 -26376.772,E2 -26376.772} C_VEL
LIN {X 0,Y 110.472,Z 219.543,A -85,B 0,C 180,E1 -26378.8,E2 -26378.8} C_VEL
LIN {X 0,Y 108.237,Z 216.062,A -85,B 0,C 180,E1 -26383.099,E2 -26383.099} C_VEL
LIN {X 0,Y 107.53,Z 210.081,A -85,B 0,C 180,E1 -26391.061,E2 -26391.061} C_VEL
LIN {X 0,Y 109.24,Z 204.235,A -85,B 0,C 180,E1 -26398.843,E2 -26398.843} C_VEL
LIN {X 0,Y 109.608,Z 202.674,A -85,B 0,C 180,E1 -26400.854,E2 -26400.854} C_VEL
LIN {X 0,Y 108.615,Z 198.96,A -85,B 0,C 180,E1 -26405.794,E2 -26405.794} C_VEL
LIN {X 0,Y 107.809,Z 199.056,A -85,B 0,C 180,E1 -26414.185,E2 -26414.185} C_VEL
LIN {X 0,Y 107.745,Z 199.064,A -85,B 0,C 180,E1 -26421.502,E2 -26421.502} C_VEL
LIN {X 0,Y 107.797,Z 199.057,A -85,B 0,C 180,E1 -26428.562,E2 -26428.562} C_VEL
LIN {X 0,Y 107.9,Z 199.043,A -85,B 0,C 180,E1 -26436.995,E2 -26436.995} C_VEL
LIN {X 0,Y 108.026,Z 199.026,A -85,B 0,C 180,E1 -26444.916,E2 -26444.916} C_VEL
LIN {X 0,Y 108.277,Z 198.997,A -85,B 0,C 180,E1 -26448.771,E2 -26448.771} C_VEL
LIN {X 0,Y 108.447,Z 198.976,A -85,B 0,C 180,E1 -26456.284,E2 -26456.284} C_VEL
LIN {X 0,Y 108.933,Z 198.907,A -85,B 0,C 180,E1 -26460,E2 -26460} C_VEL
LIN {X 0,Y 108.316,Z 198.987,A -85,B 0,C 180,E1 -26467.456,E2 -26467.456} C_VEL
LIN {X 0,Y 108.187,Z 199.009,A -85,B 0,C 180,E1 -26473.017,E2 -26473.017} C_VEL
LIN {X 0,Y 107.894,Z 199.043,A -85,B 0,C 180,E1 -26479.007,E2 -26479.007} C_VEL
LIN {X 0,Y 107.844,Z 199.047,A -85,B 0,C 180,E1 -26484.183,E2 -26484.183} C_VEL
LIN {X 0,Y 107.694,Z 199.059,A -85,B 0,C 180,E1 -26489.525,E2 -26489.525} C_VEL
LIN {X 0,Y 107.085,Z 199.146,A -85,B 0,C 180,E1 -26492.649,E2 -26492.649} C_VEL
LIN {X 0,Y 105.558,Z 199.342,A -85,B 0,C 180,E1 -26495.741,E2 -26495.741} C_VEL
LIN {X 0,Y 100.979,Z 199.91,A -85,B 0,C 180,E1 -26504.352,E2 -26504.352} C_VEL
LIN {X 0,Y 100.592,Z 199.947,A -85,B 0,C 180,E1 -26506.647,E2 -26506.647} C_VEL
LIN {X 0,Y 100.625,Z 199.944,A -85,B 0,C 180,E1 -26511.063,E2 -26511.063} C_VEL
LIN {X 0,Y 100.691,Z 199.942,A -85,B 0,C 180,E1 -26516.885,E2 -26516.885} C_VEL
LIN {X 0,Y 100.782,Z 199.93,A -85,B 0,C 180,E1 -26525.273,E2 -26525.273} C_VEL
LIN {X 0,Y 100.814,Z 199.922,A -85,B 0,C 180,E1 -26529.608,E2 -26529.608} C_VEL
LIN {X 0,Y 101.195,Z 199.873,A -85,B 0,C 180,E1 -26537.981,E2 -26537.981} C_VEL
LIN {X 0,Y 101.276,Z 199.87,A -85,B 0,C 180,E1 -26542.029,E2 -26542.029} C_VEL
LIN {X 0,Y 101.868,Z 199.797,A -85,B 0,C 180,E1 -26550.006,E2 -26550.006} C_VEL
LIN {X 0,Y 101.278,Z 199.87,A -85,B 0,C 180,E1 -26557.984,E2 -26557.984} C_VEL
LIN {X 0,Y 101.116,Z 199.882,A -85,B 0,C 180,E1 -26563.33,E2 -26563.33} C_VEL
LIN {X 0,Y 100.809,Z 199.922,A -85,B 0,C 180,E1 -26570.407,E2 -26570.407} C_VEL
LIN {X 0,Y 100.738,Z 199.936,A -85,B 0,C 180,E1 -26574.914,E2 -26574.914} C_VEL
LIN {X 0,Y 100.69,Z 199.942,A -85,B 0,C 180,E1 -26583.114,E2 -26583.114} C_VEL
LIN {X 0,Y 100.641,Z 199.944,A -85,B 0,C 180,E1 -26589.812,E2 -26589.812} C_VEL
LIN {X 0,Y 100.676,Z 199.94,A -85,B 0,C 180,E1 -26595.727,E2 -26595.727} C_VEL
LIN {X 0,Y 100.858,Z 199.921,A -85,B 0,C 180,E1 -26601.161,E2 -26601.161} C_VEL
LIN {X 0,Y 101.277,Z 199.862,A -85,B 0,C 180,E1 -26606.39,E2 -26606.39} C_VEL
LIN {X 0,Y 100.373,Z 200.116,A -85,B 0,C 180,E1 -26612.079,E2 -26612.079} C_VEL
LIN {X 0,Y 99.293,Z 204.772,A -85,B 0,C 180,E1 -26619.274,E2 -26619.274} C_VEL
LIN {X 0,Y 100.844,Z 215.506,A -85,B 0,C 180,E1 -26636.004,E2 -26636.004} C_VEL
LIN {X 0,Y 103.329,Z 218.43,A -85,B 0,C 180,E1 -26640.122,E2 -26640.122} C_VEL
LIN {X 0,Y 104.743,Z 228.766,A -85,B 0,C 180,E1 -26642.404,E2 -26642.404} C_VEL
LIN {X 0,Y 105.056,Z 240.351,A -85,B 0,C 180,E1 -26646.241,E2 -26646.241} C_VEL
LIN {X 0,Y 105.306,Z 250.285,A -85,B 0,C 180,E1 -26650.576,E2 -26650.576} C_VEL
LIN {X 0,Y 106.556,Z 261.016,A -85,B 0,C 180,E1 -26656.279,E2 -26656.279} C_VEL
LIN {X 0,Y 108.895,Z 269.749,A -85,B 0,C 180,E1 -26661.784,E2 -26661.784} C_VEL
LIN {X 0,Y 113.162,Z 278.21,A -85,B 0,C 180,E1 -26667.762,E2 -26667.762} C_VEL
LIN {X 0,Y 118.209,Z 284.338,A -85,B 0,C 180,E1 -26672.35,E2 -26672.35} C_VEL
LIN {X 0,Y 126.441,Z 290.974,A -85,B 0,C 180,E1 -26677.692,E2 -26677.692} C_VEL
LIN {X 0,Y 133.719,Z 294.986,A -85,B 0,C 180,E1 -26681.07,E2 -26681.07} C_VEL
LIN {X 0,Y 136.283,Z 296.121,A -85,B 0,C 180,E1 -26682.098,E2 -26682.098} C_VEL
LIN {X 0,Y 129.558,Z 294.331,A -85,B 0,C 180,E1 -26685.148,E2 -26685.148} C_VEL
LIN {X 0,Y 121.292,Z 291.099,A -85,B 0,C 180,E1 -26690.398,E2 -26690.398} C_VEL
LIN {X 0,Y 113.259,Z 285.755,A -85,B 0,C 180,E1 -26698.161,E2 -26698.161} C_VEL
LIN {X 0,Y 109.064,Z 280.151,A -85,B 0,C 180,E1 -26705.463,E2 -26705.463} C_VEL
LIN {X 0,Y 107.506,Z 273.802,A -85,B 0,C 180,E1 -26712.886,E2 -26712.886} C_VEL
LIN {X 0,Y 107.915,Z 266.712,A -85,B 0,C 180,E1 -26719.699,E2 -26719.699} C_VEL
LIN {X 0,Y 108.457,Z 263.11,A -85,B 0,C 180,E1 -26722.548,E2 -26722.548} C_VEL
LIN {X 0,Y 108.367,Z 260.179,A -85,B 0,C 180,E1 -26724.291,E2 -26724.291} C_VEL
LIN {X 0,Y 107.561,Z 250.884,A -85,B 0,C 180,E1 -26728.59,E2 -26728.59} C_VEL
LIN {X 0,Y 107.059,Z 240.65,A -85,B 0,C 180,E1 -26732.356,E2 -26732.356} C_VEL
LIN {X 0,Y 106.621,Z 235.691,A -85,B 0,C 180,E1 -26733.773,E2 -26733.773} C_VEL
LIN {X 0,Y 104.484,Z 222.02,A -85,B 0,C 180,E1 -26736.518,E2 -26736.518} C_VEL
LIN {X 0,Y 104.195,Z 219.449,A -85,B 0,C 180,E1 -26737.04,E2 -26737.04} C_VEL
LIN {X 0,Y 101.427,Z 215.682,A -85,B 0,C 180,E1 -26741.991,E2 -26741.991} C_VEL
LIN {X 0,Y 100.417,Z 209.773,A -85,B 0,C 180,E1 -26750.477,E2 -26750.477} C_VEL
LIN {X 0,Y 102.066,Z 204,A -85,B 0,C 180,E1 -26758.809,E2 -26758.809} C_VEL
LIN {X 0,Y 102.438,Z 202.44,A -85,B 0,C 180,E1 -26760.96,E2 -26760.96} C_VEL
LIN {X 0,Y 101.699,Z 199.821,A -85,B 0,C 180,E1 -26764.703,E2 -26764.703} C_VEL
LIN {X 0,Y 100.768,Z 199.933,A -85,B 0,C 180,E1 -26774.213,E2 -26774.213} C_VEL
LIN {X 0,Y 100.685,Z 199.943,A -85,B 0,C 180,E1 -26781.081,E2 -26781.081} C_VEL
LIN {X 0,Y 100.696,Z 199.937,A -85,B 0,C 180,E1 -26786.868,E2 -26786.868} C_VEL
LIN {X 0,Y 100.776,Z 199.926,A -85,B 0,C 180,E1 -26795.264,E2 -26795.264} C_VEL
LIN {X 0,Y 100.806,Z 199.928,A -85,B 0,C 180,E1 -26799.598,E2 -26799.598} C_VEL
LIN {X 0,Y 101.177,Z 199.881,A -85,B 0,C 180,E1 -26807.972,E2 -26807.972} C_VEL
LIN {X 0,Y 101.256,Z 199.865,A -85,B 0,C 180,E1 -26812.02,E2 -26812.02} C_VEL
LIN {X 0,Y 101.857,Z 199.789,A -85,B 0,C 180,E1 -26820,E2 -26820} C_VEL
LIN {X 0,Y 101.255,Z 199.866,A -85,B 0,C 180,E1 -26827.979,E2 -26827.979} C_VEL
LIN {X 0,Y 101.113,Z 199.889,A -85,B 0,C 180,E1 -26833.353,E2 -26833.353} C_VEL
LIN {X 0,Y 100.805,Z 199.928,A -85,B 0,C 180,E1 -26840.401,E2 -26840.401} C_VEL
LIN {X 0,Y 100.764,Z 199.927,A -85,B 0,C 180,E1 -26844.961,E2 -26844.961} C_VEL
LIN {X 0,Y 100.687,Z 199.938,A -85,B 0,C 180,E1 -26853.125,E2 -26853.125} C_VEL
LIN {X 0,Y 100.646,Z 199.947,A -85,B 0,C 180,E1 -26859.826,E2 -26859.826} C_VEL
LIN {X 0,Y 100.592,Z 199.947,A -85,B 0,C 180,E1 -26866.647,E2 -26866.647} C_VEL
LIN {X 0,Y 99.86,Z 200.042,A -85,B 0,C 180,E1 -26869.994,E2 -26869.994} C_VEL
LIN {X 0,Y 98.323,Z 200.234,A -85,B 0,C 180,E1 -26873.315,E2 -26873.315} C_VEL
LIN {X 0,Y 93.972,Z 200.783,A -85,B 0,C 180,E1 -26882.587,E2 -26882.587} C_VEL
LIN {X 0,Y 93.635,Z 200.815,A -85,B 0,C 180,E1 -26885.05,E2 -26885.05} C_VEL
LIN {X 0,Y 93.789,Z 200.803,A -85,B 0,C 180,E1 -26892.566,E2 -26892.566} C_VEL
LIN {X 0,Y 94.095,Z 200.756,A -85,B 0,C 180,E1 -26897.059,E2 -26897.059} C_VEL
LIN {X 0,Y 94.208,Z 200.75,A -85,B 0,C 180,E1 -26901.426,E2 -26901.426} C_VEL
LIN {X 0,Y 94.794,Z 200.678,A -85,B 0,C 180,E1 -26910.007,E2 -26910.007} C_VEL
LIN {X 0,Y 94.21,Z 200.75,A -85,B 0,C 180,E1 -26918.587,E2 -26918.587} C_VEL
LIN {X 0,Y 94.037,Z 200.764,A -85,B 0,C 180,E1 -26923.695,E2 -26923.695} C_VEL
LIN {X 0,Y 93.673,Z 200.81,A -85,B 0,C 180,E1 -26932.04,E2 -26932.04} C_VEL
LIN {X 0,Y 93.6,Z 200.826,A -85,B 0,C 180,E1 -26936.784,E2 -26936.784} C_VEL
LIN {X 0,Y 93.588,Z 200.827,A -85,B 0,C 180,E1 -26944.305,E2 -26944.305} C_VEL
LIN {X 0,Y 93.543,Z 200.833,A -85,B 0,C 180,E1 -26952.554,E2 -26952.554} C_VEL
LIN {X 0,Y 93.679,Z 200.811,A -85,B 0,C 180,E1 -26958.619,E2 -26958.619} C_VEL
LIN {X 0,Y 94.071,Z 200.762,A -85,B 0,C 180,E1 -26965.277,E2 -26965.277} C_VEL
LIN {X 0,Y 93.84,Z 200.796,A -85,B 0,C 180,E1 -26968.382,E2 -26968.382} C_VEL
LIN {X 0,Y 92.946,Z 201.114,A -85,B 0,C 180,E1 -26973.792,E2 -26973.792} C_VEL
LIN {X 0,Y 91.916,Z 206.109,A -85,B 0,C 180,E1 -26982.191,E2 -26982.191} C_VEL
LIN {X 0,Y 93.454,Z 214.098,A -85,B 0,C 180,E1 -26995.687,E2 -26995.687} C_VEL
LIN {X 0,Y 97.313,Z 218.609,A -85,B 0,C 180,E1 -27002.329,E2 -27002.329} C_VEL
LIN {X 0,Y 98.535,Z 226.569,A -85,B 0,C 180,E1 -27004.09,E2 -27004.09} C_VEL
LIN {X 0,Y 98.853,Z 234.395,A -85,B 0,C 180,E1 -27006.635,E2 -27006.635} C_VEL
LIN {X 0,Y 99.172,Z 242.153,A -85,B 0,C 180,E1 -27009.69,E2 -27009.69} C_VEL
LIN {X 0,Y 99.768,Z 251.545,A -85,B 0,C 180,E1 -27014.274,E2 -27014.274} C_VEL
LIN {X 0,Y 101.279,Z 260.318,A -85,B 0,C 180,E1 -27019.246,E2 -27019.246} C_VEL
LIN {X 0,Y 104.038,Z 269.031,A -85,B 0,C 180,E1 -27024.974,E2 -27024.974} C_VEL
LIN {X 0,Y 108.964,Z 277.595,A -85,B 0,C 180,E1 -27031.064,E2 -27031.064} C_VEL
LIN {X 0,Y 116.622,Z 285.669,A -85,B 0,C 180,E1 -27037.059,E2 -27037.059} C_VEL
LIN {X 0,Y 123.456,Z 290.621,A -85,B 0,C 180,E1 -27040.895,E2 -27040.895} C_VEL
LIN {X 0,Y 125.944,Z 292.101,A -85,B 0,C 180,E1 -27042.039,E2 -27042.039} C_VEL
LIN {X 0,Y 124.945,Z 291.866,A -85,B 0,C 180,E1 -27043.003,E2 -27043.003} C_VEL
LIN {X 0,Y 116.356,Z 288.246,A -85,B 0,C 180,E1 -27048.356,E2 -27048.356} C_VEL
LIN {X 0,Y 109.421,Z 283.706,A -85,B 0,C 180,E1 -27054.679,E2 -27054.679} C_VEL
LIN {X 0,Y 103.892,Z 277.122,A -85,B 0,C 180,E1 -27063.257,E2 -27063.257} C_VEL
LIN {X 0,Y 101.953,Z 269.753,A -85,B 0,C 180,E1 -27071.922,E2 -27071.922} C_VEL
LIN {X 0,Y 102.319,Z 262.624,A -85,B 0,C 180,E1 -27078.831,E2 -27078.831} C_VEL
LIN {X 0,Y 102.729,Z 259.757,A -85,B 0,C 180,E1 -27081.162,E2 -27081.162} C_VEL
LIN {X 0,Y 102.517,Z 256.42,A -85,B 0,C 180,E1 -27083.103,E2 -27083.103} C_VEL
LIN {X 0,Y 101.604,Z 246.888,A -85,B 0,C 180,E1 -27087.516,E2 -27087.516} C_VEL
LIN {X 0,Y 100.998,Z 237.322,A -85,B 0,C 180,E1 -27090.99,E2 -27090.99} C_VEL
LIN {X 0,Y 99.989,Z 231.294,A -85,B 0,C 180,E1 -27092.511,E2 -27092.511} C_VEL
LIN {X 0,Y 98.156,Z 219.466,A -85,B 0,C 180,E1 -27094.909,E2 -27094.909} C_VEL
LIN {X 0,Y 95.661,Z 216.84,A -85,B 0,C 180,E1 -27098.443,E2 -27098.443} C_VEL
LIN {X 0,Y 93.584,Z 212.454,A -85,B 0,C 180,E1 -27105.009,E2 -27105.009} C_VEL
LIN {X 0,Y 94.922,Z 203.71,A -85,B 0,C 180,E1 -27118.757,E2 -27118.757} C_VEL
LIN {X 0,Y 95.257,Z 202.154,A -85,B 0,C 180,E1 -27121.086,E2 -27121.086} C_VEL
LIN {X 0,Y 94.84,Z 200.674,A -85,B 0,C 180,E1 -27123.383,E2 -27123.383} C_VEL
LIN {X 0,Y 93.827,Z 200.797,A -85,B 0,C 180,E1 -27131.492,E2 -27131.492} C_VEL
LIN {X 0,Y 93.624,Z 200.818,A -85,B 0,C 180,E1 -27138.637,E2 -27138.637} C_VEL
LIN {X 0,Y 93.603,Z 200.817,A -85,B 0,C 180,E1 -27145.668,E2 -27145.668} C_VEL
LIN {X 0,Y 93.659,Z 200.811,A -85,B 0,C 180,E1 -27154.202,E2 -27154.202} C_VEL
LIN {X 0,Y 93.683,Z 200.816,A -85,B 0,C 180,E1 -27157.969,E2 -27157.969} C_VEL
LIN {X 0,Y 94.081,Z 200.766,A -85,B 0,C 180,E1 -27167.049,E2 -27167.049} C_VEL
LIN {X 0,Y 94.189,Z 200.745,A -85,B 0,C 180,E1 -27171.417,E2 -27171.417} C_VEL
LIN {X 0,Y 94.783,Z 200.67,A -85,B 0,C 180,E1 -27180,E2 -27180} C_VEL
LIN {X 0,Y 94.188,Z 200.745,A -85,B 0,C 180,E1 -27188.582,E2 -27188.582} C_VEL
LIN {X 0,Y 94.031,Z 200.772,A -85,B 0,C 180,E1 -27193.71,E2 -27193.71} C_VEL
LIN {X 0,Y 93.682,Z 200.816,A -85,B 0,C 180,E1 -27202.03,E2 -27202.03} C_VEL
LIN {X 0,Y 93.61,Z 200.819,A -85,B 0,C 180,E1 -27206.773,E2 -27206.773} C_VEL
LIN {X 0,Y 93.587,Z 200.82,A -85,B 0,C 180,E1 -27214.317,E2 -27214.317} C_VEL
LIN {X 0,Y 93.531,Z 200.826,A -85,B 0,C 180,E1 -27222.552,E2 -27222.552} C_VEL
LIN {X 0,Y 93.531,Z 200.834,A -85,B 0,C 180,E1 -27228.712,E2 -27228.712} C_VEL
LIN {X 0,Y 93.587,Z 200.827,A -85,B 0,C 180,E1 -27235.696,E2 -27235.696} C_VEL
LIN {X 0,Y 93.664,Z 200.818,A -85,B 0,C 180,E1 -27244.211,E2 -27244.211} C_VEL
LIN {X 0,Y 93.635,Z 200.815,A -85,B 0,C 180,E1 -27245.05,E2 -27245.05} C_VEL
LIN {X 0,Y 92.929,Z 200.904,A -85,B 0,C 180,E1 -27248.647,E2 -27248.647} C_VEL
LIN {X 0,Y 91.396,Z 201.1,A -85,B 0,C 180,E1 -27252.219,E2 -27252.219} C_VEL
LIN {X 0,Y 87.316,Z 201.608,A -85,B 0,C 180,E1 -27262.25,E2 -27262.25} C_VEL
LIN {X 0,Y 87.19,Z 201.614,A -85,B 0,C 180,E1 -27264.904,E2 -27264.904} C_VEL
LIN {X 0,Y 87.722,Z 201.559,A -85,B 0,C 180,E1 -27270.007,E2 -27270.007} C_VEL
LIN {X 0,Y 87.115,Z 201.634,A -85,B 0,C 180,E1 -27279.293,E2 -27279.293} C_VEL
LIN {X 0,Y 86.953,Z 201.648,A -85,B 0,C 180,E1 -27284.094,E2 -27284.094} C_VEL
LIN {X 0,Y 86.567,Z 201.701,A -85,B 0,C 180,E1 -27293.957,E2 -27293.957} C_VEL
LIN {X 0,Y 86.462,Z 201.707,A -85,B 0,C 180,E1 -27299.198,E2 -27299.198} C_VEL
LIN {X 0,Y 86.507,Z 201.708,A -85,B 0,C 180,E1 -27305.667,E2 -27305.667} C_VEL
LIN {X 0,Y 86.492,Z 201.711,A -85,B 0,C 180,E1 -27313.004,E2 -27313.004} C_VEL
LIN {X 0,Y 86.641,Z 201.69,A -85,B 0,C 180,E1 -27319.539,E2 -27319.539} C_VEL
LIN {X 0,Y 86.983,Z 201.643,A -85,B 0,C 180,E1 -27325.558,E2 -27325.558} C_VEL
LIN {X 0,Y 86.306,Z 201.735,A -85,B 0,C 180,E1 -27330.752,E2 -27330.752} C_VEL
LIN {X 0,Y 85.536,Z 202.035,A -85,B 0,C 180,E1 -27335.744,E2 -27335.744} C_VEL
LIN {X 0,Y 84.832,Z 208.695,A -85,B 0,C 180,E1 -27348.047,E2 -27348.047} C_VEL
LIN {X 0,Y 86.963,Z 214.051,A -85,B 0,C 180,E1 -27357.685,E2 -27357.685} C_VEL
LIN {X 0,Y 91.506,Z 218.572,A -85,B 0,C 180,E1 -27364.815,E2 -27364.815} C_VEL
LIN {X 0,Y 92.723,Z 226.255,A -85,B 0,C 180,E1 -27366.611,E2 -27366.611} C_VEL
LIN {X 0,Y 93.342,Z 236.894,A -85,B 0,C 180,E1 -27370.466,E2 -27370.466} C_VEL
LIN {X 0,Y 93.935,Z 246.774,A -85,B 0,C 180,E1 -27375.181,E2 -27375.181} C_VEL
LIN {X 0,Y 95.876,Z 257.853,A -85,B 0,C 180,E1 -27381.501,E2 -27381.501} C_VEL
LIN {X 0,Y 98.946,Z 266.825,A -85,B 0,C 180,E1 -27387.496,E2 -27387.496} C_VEL
LIN {X 0,Y 104.303,Z 275.689,A -85,B 0,C 180,E1 -27393.772,E2 -27393.772} C_VEL
LIN {X 0,Y 111.326,Z 283.17,A -85,B 0,C 180,E1 -27399.147,E2 -27399.147} C_VEL
LIN {X 0,Y 116.785,Z 287.454,A -85,B 0,C 180,E1 -27402.293,E2 -27402.293} C_VEL
LIN {X 0,Y 115.909,Z 287.189,A -85,B 0,C 180,E1 -27403.307,E2 -27403.307} C_VEL
LIN {X 0,Y 106.088,Z 281.545,A -85,B 0,C 180,E1 -27410.991,E2 -27410.991} C_VEL
LIN {X 0,Y 100.511,Z 276.084,A -85,B 0,C 180,E1 -27418.128,E2 -27418.128} C_VEL
LIN {X 0,Y 97.132,Z 269.235,A -85,B 0,C 180,E1 -27426.543,E2 -27426.543} C_VEL
LIN {X 0,Y 96.505,Z 262.253,A -85,B 0,C 180,E1 -27434.142,E2 -27434.142} C_VEL
LIN {X 0,Y 97.136,Z 256.867,A -85,B 0,C 180,E1 -27439.092,E2 -27439.092} C_VEL
LIN {X 0,Y 97.031,Z 254.231,A -85,B 0,C 180,E1 -27440.805,E2 -27440.805} C_VEL
LIN {X 0,Y 95.972,Z 245.002,A -85,B 0,C 180,E1 -27445.268,E2 -27445.268} C_VEL
LIN {X 0,Y 95.133,Z 235.252,A -85,B 0,C 180,E1 -27448.935,E2 -27448.935} C_VEL
LIN {X 0,Y 93.029,Z 224.186,A -85,B 0,C 180,E1 -27451.468,E2 -27451.468} C_VEL
LIN {X 0,Y 92.315,Z 219.42,A -85,B 0,C 180,E1 -27452.471,E2 -27452.471} C_VEL
LIN {X 0,Y 89.107,Z 216.389,A -85,B 0,C 180,E1 -27456.787,E2 -27456.787} C_VEL
LIN {X 0,Y 86.354,Z 210.452,A -85,B 0,C 180,E1 -27466.542,E2 -27466.542} C_VEL
LIN {X 0,Y 87.757,Z 203.37,A -85,B 0,C 180,E1 -27478.71,E2 -27478.71} C_VEL
LIN {X 0,Y 87.991,Z 201.525,A -85,B 0,C 180,E1 -27481.771,E2 -27481.771} C_VEL
LIN {X 0,Y 87.358,Z 201.604,A -85,B 0,C 180,E1 -27486.437,E2 -27486.437} C_VEL
LIN {X 0,Y 86.591,Z 201.69,A -85,B 0,C 180,E1 -27496.914,E2 -27496.914} C_VEL
LIN {X 0,Y 86.551,Z 201.696,A -85,B 0,C 180,E1 -27505.36,E2 -27505.36} C_VEL
LIN {X 0,Y 86.574,Z 201.695,A -85,B 0,C 180,E1 -27513.231,E2 -27513.231} C_VEL
LIN {X 0,Y 86.636,Z 201.689,A -85,B 0,C 180,E1 -27521.065,E2 -27521.065} C_VEL
LIN {X 0,Y 86.959,Z 201.653,A -85,B 0,C 180,E1 -27525.968,E2 -27525.968} C_VEL
LIN {X 0,Y 87.097,Z 201.629,A -85,B 0,C 180,E1 -27530.712,E2 -27530.712} C_VEL
LIN {X 0,Y 87.71,Z 201.55,A -85,B 0,C 180,E1 -27540,E2 -27540} C_VEL
LIN {X 0,Y 87.096,Z 201.629,A -85,B 0,C 180,E1 -27549.287,E2 -27549.287} C_VEL
LIN {X 0,Y 86.939,Z 201.655,A -85,B 0,C 180,E1 -27554.089,E2 -27554.089} C_VEL
LIN {X 0,Y 86.576,Z 201.696,A -85,B 0,C 180,E1 -27563.946,E2 -27563.946} C_VEL
LIN {X 0,Y 86.465,Z 201.714,A -85,B 0,C 180,E1 -27569.188,E2 -27569.188} C_VEL
LIN {X 0,Y 86.506,Z 201.704,A -85,B 0,C 180,E1 -27575.68,E2 -27575.68} C_VEL
LIN {X 0,Y 86.473,Z 201.705,A -85,B 0,C 180,E1 -27583.002,E2 -27583.002} C_VEL
LIN {X 0,Y 86.453,Z 201.712,A -85,B 0,C 180,E1 -27589.443,E2 -27589.443} C_VEL
LIN {X 0,Y 86.53,Z 201.707,A -85,B 0,C 180,E1 -27595.361,E2 -27595.361} C_VEL
LIN {X 0,Y 86.58,Z 201.7,A -85,B 0,C 180,E1 -27603.24,E2 -27603.24} C_VEL
LIN {X 0,Y 86.644,Z 201.69,A -85,B 0,C 180,E1 -27611.075,E2 -27611.075} C_VEL
LIN {X 0,Y 86.967,Z 201.646,A -85,B 0,C 180,E1 -27615.977,E2 -27615.977} C_VEL
LIN {X 0,Y 87.114,Z 201.634,A -85,B 0,C 180,E1 -27620.722,E2 -27620.722} C_VEL
LIN {X 0,Y 87.19,Z 201.614,A -85,B 0,C 180,E1 -27624.904,E2 -27624.904} C_VEL
LIN {X 0,Y 87.023,Z 201.645,A -85,B 0,C 180,E1 -27627.479,E2 -27627.479} C_VEL
LIN {X 0,Y 85.784,Z 201.813,A -85,B 0,C 180,E1 -27631.312,E2 -27631.312} C_VEL
LIN {X 0,Y 82.501,Z 202.229,A -85,B 0,C 180,E1 -27637.802,E2 -27637.802} C_VEL
LIN {X 0,Y 80.216,Z 202.499,A -85,B 0,C 180,E1 -27643.375,E2 -27643.375} C_VEL
LIN {X 0,Y 79.665,Z 202.552,A -85,B 0,C 180,E1 -27646.296,E2 -27646.296} C_VEL
LIN {X 0,Y 79.503,Z 202.574,A -85,B 0,C 180,E1 -27650.716,E2 -27650.716} C_VEL
LIN {X 0,Y 79.468,Z 202.583,A -85,B 0,C 180,E1 -27657.825,E2 -27657.825} C_VEL
LIN {X 0,Y 79.373,Z 202.595,A -85,B 0,C 180,E1 -27662.1,E2 -27662.1} C_VEL
LIN {X 0,Y 79.369,Z 202.59,A -85,B 0,C 180,E1 -27668.314,E2 -27668.314} C_VEL
LIN {X 0,Y 79.449,Z 202.585,A -85,B 0,C 180,E1 -27675.057,E2 -27675.057} C_VEL
LIN {X 0,Y 79.702,Z 202.556,A -85,B 0,C 180,E1 -27682.536,E2 -27682.536} C_VEL
LIN {X 0,Y 79.518,Z 202.579,A -85,B 0,C 180,E1 -27687.975,E2 -27687.975} C_VEL
LIN {X 0,Y 78.779,Z 202.668,A -85,B 0,C 180,E1 -27693.509,E2 -27693.509} C_VEL
LIN {X 0,Y 78.118,Z 202.978,A -85,B 0,C 180,E1 -27698.216,E2 -27698.216} C_VEL
LIN {X 0,Y 80.611,Z 213.949,A -85,B 0,C 180,E1 -27720,E2 -27720} C_VEL
LIN {X 0,Y 85.61,Z 218.396,A -85,B 0,C 180,E1 -27727.358,E2 -27727.358} C_VEL
LIN {X 0,Y 86.005,Z 218.65,A -85,B 0,C 180,E1 -27727.714,E2 -27727.714} C_VEL
LIN {X 0,Y 87.1,Z 225.12,A -85,B 0,C 180,E1 -27729.287,E2 -27729.287} C_VEL
LIN {X 0,Y 87.843,Z 235.241,A -85,B 0,C 180,E1 -27733.148,E2 -27733.148} C_VEL
LIN {X 0,Y 88.636,Z 244.738,A -85,B 0,C 180,E1 -27737.898,E2 -27737.898} C_VEL
LIN {X 0,Y 90.721,Z 255.148,A -85,B 0,C 180,E1 -27743.999,E2 -27743.999} C_VEL
LIN {X 0,Y 94.864,Z 265.85,A -85,B 0,C 180,E1 -27751.238,E2 -27751.238} C_VEL
LIN {X 0,Y 100.917,Z 274.801,A -85,B 0,C 180,E1 -27757.544,E2 -27757.544} C_VEL
LIN {X 0,Y 108.165,Z 282.028,A -85,B 0,C 180,E1 -27762.572,E2 -27762.572} C_VEL
LIN {X 0,Y 107.284,Z 281.719,A -85,B 0,C 180,E1 -27763.889,E2 -27763.889} C_VEL
LIN {X 0,Y 99.283,Z 276.077,A -85,B 0,C 180,E1 -27771.139,E2 -27771.139} C_VEL
LIN {X 0,Y 93.374,Z 268.519,A -85,B 0,C 180,E1 -27780.702,E2 -27780.702} C_VEL
LIN {X 0,Y 91.391,Z 260.544,A -85,B 0,C 180,E1 -27790.066,E2 -27790.066} C_VEL
LIN {X 0,Y 91.723,Z 253.866,A -85,B 0,C 180,E1 -27796.704,E2 -27796.704} C_VEL
LIN {X 0,Y 91.848,Z 252.481,A -85,B 0,C 180,E1 -27797.846,E2 -27797.846} C_VEL
LIN {X 0,Y 90.828,Z 245.275,A -85,B 0,C 180,E1 -27801.651,E2 -27801.651} C_VEL
LIN {X 0,Y 89.809,Z 236.087,A -85,B 0,C 180,E1 -27805.505,E2 -27805.505} C_VEL
LIN {X 0,Y 89.12,Z 231.676,A -85,B 0,C 180,E1 -27806.885,E2 -27806.885} C_VEL
LIN {X 0,Y 86.664,Z 219.339,A -85,B 0,C 180,E1 -27809.702,E2 -27809.702} C_VEL
LIN {X 0,Y 82.637,Z 215.9,A -85,B 0,C 180,E1 -27814.871,E2 -27814.871} C_VEL
LIN {X 0,Y 79.427,Z 210.018,A -85,B 0,C 180,E1 -27825.385,E2 -27825.385} C_VEL
LIN {X 0,Y 80.79,Z 202.418,A -85,B 0,C 180,E1 -27839.857,E2 -27839.857} C_VEL
LIN {X 0,Y 80.982,Z 202.397,A -85,B 0,C 180,E1 -27841.37,E2 -27841.37} C_VEL
LIN {X 0,Y 80.073,Z 202.505,A -85,B 0,C 180,E1 -27847.897,E2 -27847.897} C_VEL
LIN {X 0,Y 79.568,Z 202.571,A -85,B 0,C 180,E1 -27855.039,E2 -27855.039} C_VEL
LIN {X 0,Y 79.444,Z 202.588,A -85,B 0,C 180,E1 -27862.753,E2 -27862.753} C_VEL
LIN {X 0,Y 79.473,Z 202.582,A -85,B 0,C 180,E1 -27872.15,E2 -27872.15} C_VEL
LIN {X 0,Y 79.503,Z 202.582,A -85,B 0,C 180,E1 -27879.292,E2 -27879.292} C_VEL
LIN {X 0,Y 79.83,Z 202.539,A -85,B 0,C 180,E1 -27885.524,E2 -27885.524} C_VEL
LIN {X 0,Y 79.982,Z 202.517,A -85,B 0,C 180,E1 -27889.878,E2 -27889.878} C_VEL
LIN {X 0,Y 80.638,Z 202.431,A -85,B 0,C 180,E1 -27900,E2 -27900} C_VEL
LIN {X 0,Y 79.981,Z 202.517,A -85,B 0,C 180,E1 -27910.121,E2 -27910.121} C_VEL
LIN {X 0,Y 79.751,Z 202.547,A -85,B 0,C 180,E1 -27915.329,E2 -27915.329} C_VEL
LIN {X 0,Y 79.503,Z 202.582,A -85,B 0,C 180,E1 -27920.707,E2 -27920.707} C_VEL
LIN {X 0,Y 79.471,Z 202.582,A -85,B 0,C 180,E1 -27927.847,E2 -27927.847} C_VEL
LIN {X 0,Y 79.373,Z 202.595,A -85,B 0,C 180,E1 -27932.091,E2 -27932.091} C_VEL
LIN {X 0,Y 79.363,Z 202.599,A -85,B 0,C 180,E1 -27938.307,E2 -27938.307} C_VEL
LIN {X 0,Y 79.402,Z 202.591,A -85,B 0,C 180,E1 -27945.08,E2 -27945.08} C_VEL
LIN {X 0,Y 79.382,Z 202.591,A -85,B 0,C 180,E1 -27952.826,E2 -27952.826} C_VEL
LIN {X 0,Y 79.375,Z 202.595,A -85,B 0,C 180,E1 -27957.92,E2 -27957.92} C_VEL
LIN {X 0,Y 79.521,Z 202.579,A -85,B 0,C 180,E1 -27963.784,E2 -27963.784} C_VEL
LIN {X 0,Y 79.51,Z 202.573,A -85,B 0,C 180,E1 -27969.303,E2 -27969.303} C_VEL
LIN {X 0,Y 79.839,Z 202.535,A -85,B 0,C 180,E1 -27975.534,E2 -27975.534} C_VEL
LIN {X 0,Y 79.997,Z 202.518,A -85,B 0,C 180,E1 -27979.888,E2 -27979.888} C_VEL
LIN {X 0,Y 80.651,Z 202.44,A -85,B 0,C 180,E1 -27990.008,E2 -27990.008} C_VEL
LIN {X 0,Y 79.994,Z 202.519,A -85,B 0,C 180,E1 -28000.128,E2 -28000.128} C_VEL
LIN {X 0,Y 79.665,Z 202.552,A -85,B 0,C 180,E1 -28006.296,E2 -28006.296} C_VEL
LIN {X 0,Y 78.741,Z 202.671,A -85,B 0,C 180,E1 -28010.515,E2 -28010.515} C_VEL
LIN {X 0,Y 77.096,Z 202.881,A -85,B 0,C 180,E1 -28014.717,E2 -28014.717} C_VEL
LIN {X 0,Y 72.268,Z 203.473,A -85,B 0,C 180,E1 -28029.832,E2 -28029.832} C_VEL
LIN {X 0,Y 72.355,Z 203.463,A -85,B 0,C 180,E1 -28037.162,E2 -28037.162} C_VEL
LIN {X 0,Y 72.504,Z 203.454,A -85,B 0,C 180,E1 -28040.86,E2 -28040.86} C_VEL
LIN {X 0,Y 72.514,Z 203.447,A -85,B 0,C 180,E1 -28044.443,E2 -28044.443} C_VEL
LIN {X 0,Y 71.911,Z 203.528,A -85,B 0,C 180,E1 -28051.61,E2 -28051.61} C_VEL
LIN {X 0,Y 70.773,Z 203.848,A -85,B 0,C 180,E1 -28061.172,E2 -28061.172} C_VEL
LIN {X 0,Y 73.209,Z 212.42,A -85,B 0,C 180,E1 -28080,E2 -28080} C_VEL
LIN {X 0,Y 78.139,Z 216.916,A -85,B 0,C 180,E1 -28088.314,E2 -28088.314} C_VEL
LIN {X 0,Y 80.762,Z 218.671,A -85,B 0,C 180,E1 -28091.057,E2 -28091.057} C_VEL
LIN {X 0,Y 81.732,Z 223.505,A -85,B 0,C 180,E1 -28092.242,E2 -28092.242} C_VEL
LIN {X 0,Y 82.624,Z 233.388,A -85,B 0,C 180,E1 -28096.175,E2 -28096.175} C_VEL
LIN {X 0,Y 83.875,Z 243.848,A -85,B 0,C 180,E1 -28101.699,E2 -28101.699} C_VEL
LIN {X 0,Y 86.43,Z 253.928,A -85,B 0,C 180,E1 -28107.876,E2 -28107.876} C_VEL
LIN {X 0,Y 90.462,Z 263.26,A -85,B 0,C 180,E1 -28114.282,E2 -28114.282} C_VEL
LIN {X 0,Y 96.968,Z 272.566,A -85,B 0,C 180,E1 -28120.715,E2 -28120.715} C_VEL
LIN {X 0,Y 99.181,Z 274.956,A -85,B 0,C 180,E1 -28122.313,E2 -28122.313} C_VEL
LIN {X 0,Y 100.244,Z 276.199,A -85,B 0,C 180,E1 -28123.701,E2 -28123.701} C_VEL
LIN {X 0,Y 92.143,Z 269.272,A -85,B 0,C 180,E1 -28132.389,E2 -28132.389} C_VEL
LIN {X 0,Y 87.565,Z 261.575,A -85,B 0,C 180,E1 -28141.991,E2 -28141.991} C_VEL
LIN {X 0,Y 86.388,Z 253.652,A -85,B 0,C 180,E1 -28151.002,E2 -28151.002} C_VEL
LIN {X 0,Y 86.651,Z 249.959,A -85,B 0,C 180,E1 -28154.709,E2 -28154.709} C_VEL
LIN {X 0,Y 86.49,Z 247.465,A -85,B 0,C 180,E1 -28156.483,E2 -28156.483} C_VEL
LIN {X 0,Y 85.054,Z 238.045,A -85,B 0,C 180,E1 -28161.08,E2 -28161.08} C_VEL
LIN {X 0,Y 84.233,Z 232.019,A -85,B 0,C 180,E1 -28163.405,E2 -28163.405} C_VEL
LIN {X 0,Y 81.385,Z 219.291,A -85,B 0,C 180,E1 -28166.434,E2 -28166.434} C_VEL
LIN {X 0,Y 76.096,Z 215.156,A -85,B 0,C 180,E1 -28172.968,E2 -28172.968} C_VEL
LIN {X 0,Y 72.502,Z 209.419,A -85,B 0,C 180,E1 -28184.22,E2 -28184.22} C_VEL
LIN {X 0,Y 73.124,Z 203.377,A -85,B 0,C 180,E1 -28197.153,E2 -28197.153} C_VEL
LIN {X 0,Y 73.894,Z 203.278,A -85,B 0,C 180,E1 -28201.13,E2 -28201.13} C_VEL
LIN {X 0,Y 72.562,Z 203.447,A -85,B 0,C 180,E1 -28212.674,E2 -28212.674} C_VEL
LIN {X 0,Y 72.369,Z 203.471,A -85,B 0,C 180,E1 -28220.963,E2 -28220.963} C_VEL
LIN {X 0,Y 72.329,Z 203.469,A -85,B 0,C 180,E1 -28224.337,E2 -28224.337} C_VEL
LIN {X 0,Y 72.382,Z 203.468,A -85,B 0,C 180,E1 -28230.956,E2 -28230.956} C_VEL
LIN {X 0,Y 72.384,Z 203.467,A -85,B 0,C 180,E1 -28237.146,E2 -28237.146} C_VEL
LIN {X 0,Y 72.725,Z 203.423,A -85,B 0,C 180,E1 -28245.064,E2 -28245.064} C_VEL
LIN {X 0,Y 72.869,Z 203.406,A -85,B 0,C 180,E1 -28248.878,E2 -28248.878} C_VEL
LIN {X 0,Y 73.565,Z 203.312,A -85,B 0,C 180,E1 -28260,E2 -28260} C_VEL
LIN {X 0,Y 72.868,Z 203.406,A -85,B 0,C 180,E1 -28271.121,E2 -28271.121} C_VEL
LIN {X 0,Y 72.571,Z 203.436,A -85,B 0,C 180,E1 -28276.889,E2 -28276.889} C_VEL
LIN {X 0,Y 72.383,Z 203.467,A -85,B 0,C 180,E1 -28282.853,E2 -28282.853} C_VEL
LIN {X 0,Y 72.366,Z 203.47,A -85,B 0,C 180,E1 -28289.086,E2 -28289.086} C_VEL
LIN {X 0,Y 72.29,Z 203.474,A -85,B 0,C 180,E1 -28295.684,E2 -28295.684} C_VEL
LIN {X 0,Y 72.253,Z 203.476,A -85,B 0,C 180,E1 -28302.912,E2 -28302.912} C_VEL
LIN {X 0,Y 72.29,Z 203.472,A -85,B 0,C 180,E1 -28311.055,E2 -28311.055} C_VEL
LIN {X 0,Y 72.29,Z 203.479,A -85,B 0,C 180,E1 -28314.327,E2 -28314.327} C_VEL
LIN {X 0,Y 72.369,Z 203.462,A -85,B 0,C 180,E1 -28320.961,E2 -28320.961} C_VEL
LIN {X 0,Y 72.39,Z 203.462,A -85,B 0,C 180,E1 -28327.159,E2 -28327.159} C_VEL
LIN {X 0,Y 72.734,Z 203.422,A -85,B 0,C 180,E1 -28335.074,E2 -28335.074} C_VEL
LIN {X 0,Y 72.882,Z 203.401,A -85,B 0,C 180,E1 -28338.889,E2 -28338.889} C_VEL
LIN {X 0,Y 73.578,Z 203.321,A -85,B 0,C 180,E1 -28350.009,E2 -28350.009} C_VEL
LIN {X 0,Y 72.881,Z 203.401,A -85,B 0,C 180,E1 -28361.129,E2 -28361.129} C_VEL
LIN {X 0,Y 72.581,Z 203.444,A -85,B 0,C 180,E1 -28366.896,E2 -28366.896} C_VEL
LIN {X 0,Y 72.383,Z 203.463,A -85,B 0,C 180,E1 -28372.863,E2 -28372.863} C_VEL
LIN {X 0,Y 72.363,Z 203.463,A -85,B 0,C 180,E1 -28379.062,E2 -28379.062} C_VEL
LIN {X 0,Y 72.295,Z 203.478,A -85,B 0,C 180,E1 -28385.691,E2 -28385.691} C_VEL
LIN {X 0,Y 72.268,Z 203.473,A -85,B 0,C 180,E1 -28389.832,E2 -28389.832} C_VEL
LIN {X 0,Y 71.885,Z 203.531,A -85,B 0,C 180,E1 -28392.951,E2 -28392.951} C_VEL
LIN {X 0,Y 70.499,Z 203.698,A -85,B 0,C 180,E1 -28397.599,E2 -28397.599} C_VEL
LIN {X 0,Y 68.586,Z 203.941,A -85,B 0,C 180,E1 -28402.268,E2 -28402.268} C_VEL
LIN {X 0,Y 64.137,Z 204.482,A -85,B 0,C 180,E1 -28415.995,E2 -28415.995} C_VEL
LIN {X 0,Y 63.614,Z 204.647,A -85,B 0,C 180,E1 -28424.789,E2 -28424.789} C_VEL
LIN {X 0,Y 67.026,Z 212.21,A -85,B 0,C 180,E1 -28443.006,E2 -28443.006} C_VEL
LIN {X 0,Y 72.19,Z 216.424,A -85,B 0,C 180,E1 -28451.228,E2 -28451.228} C_VEL
LIN {X 0,Y 75.987,Z 218.75,A -85,B 0,C 180,E1 -28454.907,E2 -28454.907} C_VEL
LIN {X 0,Y 76.786,Z 222.602,A -85,B 0,C 180,E1 -28455.937,E2 -28455.937} C_VEL
LIN {X 0,Y 77.784,Z 231.299,A -85,B 0,C 180,E1 -28459.577,E2 -28459.577} C_VEL
LIN {X 0,Y 79.326,Z 241.484,A -85,B 0,C 180,E1 -28465.154,E2 -28465.154} C_VEL
LIN {X 0,Y 81.969,Z 250.814,A -85,B 0,C 180,E1 -28470.961,E2 -28470.961} C_VEL
LIN {X 0,Y 86.414,Z 260.445,A -85,B 0,C 180,E1 -28477.588,E2 -28477.588} C_VEL
LIN {X 0,Y 92.869,Z 269.456,A -85,B 0,C 180,E1 -28483.693,E2 -28483.693} C_VEL
LIN {X 0,Y 92.32,Z 269.127,A -85,B 0,C 180,E1 -28484.802,E2 -28484.802} C_VEL
LIN {X 0,Y 85.141,Z 261.178,A -85,B 0,C 180,E1 -28494.694,E2 -28494.694} C_VEL
LIN {X 0,Y 82.086,Z 253.122,A -85,B 0,C 180,E1 -28504.645,E2 -28504.645} C_VEL
LIN {X 0,Y 81.852,Z 245.816,A -85,B 0,C 180,E1 -28512.501,E2 -28512.501} C_VEL
LIN {X 0,Y 81.436,Z 242.95,A -85,B 0,C 180,E1 -28514.346,E2 -28514.346} C_VEL
LIN {X 0,Y 79.912,Z 234.151,A -85,B 0,C 180,E1 -28518.579,E2 -28518.579} C_VEL
LIN {X 0,Y 79.171,Z 230.074,A -85,B 0,C 180,E1 -28520.069,E2 -28520.069} C_VEL
LIN {X 0,Y 76.633,Z 219.319,A -85,B 0,C 180,E1 -28522.58,E2 -28522.58} C_VEL
LIN {X 0,Y 72.135,Z 216.414,A -85,B 0,C 180,E1 -28527.057,E2 -28527.057} C_VEL
LIN {X 0,Y 67.287,Z 211.818,A -85,B 0,C 180,E1 -28535.986,E2 -28535.986} C_VEL
LIN {X 0,Y 65.426,Z 204.405,A -85,B 0,C 180,E1 -28553.115,E2 -28553.115} C_VEL
LIN {X 0,Y 66.672,Z 204.178,A -85,B 0,C 180,E1 -28561.795,E2 -28561.795} C_VEL
LIN {X 0,Y 65.572,Z 204.315,A -85,B 0,C 180,E1 -28571.386,E2 -28571.386} C_VEL
LIN {X 0,Y 65.295,Z 204.35,A -85,B 0,C 180,E1 -28579.773,E2 -28579.773} C_VEL
LIN {X 0,Y 65.251,Z 204.357,A -85,B 0,C 180,E1 -28589.483,E2 -28589.483} C_VEL
LIN {X 0,Y 65.235,Z 204.35,A -85,B 0,C 180,E1 -28594.473,E2 -28594.473} C_VEL
LIN {X 0,Y 65.625,Z 204.305,A -85,B 0,C 180,E1 -28604.505,E2 -28604.505} C_VEL
LIN {X 0,Y 65.762,Z 204.293,A -85,B 0,C 180,E1 -28607.658,E2 -28607.658} C_VEL
LIN {X 0,Y 66.489,Z 204.193,A -85,B 0,C 180,E1 -28620,E2 -28620} C_VEL
LIN {X 0,Y 65.761,Z 204.293,A -85,B 0,C 180,E1 -28632.341,E2 -28632.341} C_VEL
LIN {X 0,Y 65.374,Z 204.336,A -85,B 0,C 180,E1 -28638.814,E2 -28638.814} C_VEL
LIN {X 0,Y 65.227,Z 204.351,A -85,B 0,C 180,E1 -28645.53,E2 -28645.53} C_VEL
LIN {X 0,Y 65.188,Z 204.359,A -85,B 0,C 180,E1 -28652.619,E2 -28652.619} C_VEL
LIN {X 0,Y 65.184,Z 204.36,A -85,B 0,C 180,E1 -28661.015,E2 -28661.015} C_VEL
LIN {X 0,Y 65.202,Z 204.358,A -85,B 0,C 180,E1 -28669.718,E2 -28669.718} C_VEL
LIN {X 0,Y 65.248,Z 204.348,A -85,B 0,C 180,E1 -28679.507,E2 -28679.507} C_VEL
LIN {X 0,Y 65.235,Z 204.36,A -85,B 0,C 180,E1 -28684.484,E2 -28684.484} C_VEL
LIN {X 0,Y 65.634,Z 204.307,A -85,B 0,C 180,E1 -28694.516,E2 -28694.516} C_VEL
LIN {X 0,Y 65.773,Z 204.283,A -85,B 0,C 180,E1 -28697.67,E2 -28697.67} C_VEL
LIN {X 0,Y 66.502,Z 204.202,A -85,B 0,C 180,E1 -28710.01,E2 -28710.01} C_VEL
LIN {X 0,Y 65.781,Z 204.282,A -85,B 0,C 180,E1 -28722.348,E2 -28722.348} C_VEL
LIN {X 0,Y 65.38,Z 204.339,A -85,B 0,C 180,E1 -28728.823,E2 -28728.823} C_VEL
LIN {X 0,Y 65.228,Z 204.36,A -85,B 0,C 180,E1 -28735.54,E2 -28735.54} C_VEL
LIN {X 0,Y 65.173,Z 204.365,A -85,B 0,C 180,E1 -28742.639,E2 -28742.639} C_VEL
LIN {X 0,Y 65.206,Z 204.36,A -85,B 0,C 180,E1 -28751.021,E2 -28751.021} C_VEL
LIN {X 0,Y 65.381,Z 204.339,A -85,B 0,C 180,E1 -28759.838,E2 -28759.838} C_VEL
LIN {X 0,Y 65.109,Z 204.369,A -85,B 0,C 180,E1 -28767.336,E2 -28767.336} C_VEL
LIN {X 0,Y 64.987,Z 204.392,A -85,B 0,C 180,E1 -28769.919,E2 -28769.919} C_VEL
LIN {X 0,Y 64.137,Z 204.482,A -85,B 0,C 180,E1 -28775.995,E2 -28775.995} C_VEL
LIN {X 0,Y 63.097,Z 204.629,A -85,B 0,C 180,E1 -28779.467,E2 -28779.467} C_VEL
LIN {X 0,Y 60.04,Z 205.082,A -85,B 0,C 180,E1 -28785.078,E2 -28785.078} C_VEL
LIN {X 0,Y 57.504,Z 206.248,A -85,B 0,C 180,E1 -28791.117,E2 -28791.117} C_VEL
LIN {X 0,Y 57.34,Z 207.406,A -85,B 0,C 180,E1 -28794.941,E2 -28794.941} C_VEL
LIN {X 0,Y 62.779,Z 213.345,A -85,B 0,C 180,E1 -28809.668,E2 -28809.668} C_VEL
LIN {X 0,Y 69.48,Z 217.638,A -85,B 0,C 180,E1 -28817.666,E2 -28817.666} C_VEL
LIN {X 0,Y 71.683,Z 218.792,A -85,B 0,C 180,E1 -28819.324,E2 -28819.324} C_VEL
LIN {X 0,Y 72.408,Z 222.67,A -85,B 0,C 180,E1 -28820.601,E2 -28820.601} C_VEL
LIN {X 0,Y 73.568,Z 230.583,A -85,B 0,C 180,E1 -28824.221,E2 -28824.221} C_VEL
LIN {X 0,Y 75.902,Z 241.606,A -85,B 0,C 180,E1 -28830.615,E2 -28830.615} C_VEL
LIN {X 0,Y 79.484,Z 251.279,A -85,B 0,C 180,E1 -28836.945,E2 -28836.945} C_VEL
LIN {X 0,Y 84.741,Z 260.432,A -85,B 0,C 180,E1 -28843.174,E2 -28843.174} C_VEL
LIN {X 0,Y 85.794,Z 261.889,A -85,B 0,C 180,E1 -28844.131,E2 -28844.131} C_VEL
LIN {X 0,Y 83.818,Z 260.045,A -85,B 0,C 180,E1 -28847.863,E2 -28847.863} C_VEL
LIN {X 0,Y 78.94,Z 252.207,A -85,B 0,C 180,E1 -28857.703,E2 -28857.703} C_VEL
LIN {X 0,Y 77.345,Z 244.215,A -85,B 0,C 180,E1 -28867.133,E2 -28867.133} C_VEL
LIN {X 0,Y 77.305,Z 241.312,A -85,B 0,C 180,E1 -28870.102,E2 -28870.102} C_VEL
LIN {X 0,Y 75.833,Z 234.269,A -85,B 0,C 180,E1 -28873.849,E2 -28873.849} C_VEL
LIN {X 0,Y 75.011,Z 229.796,A -85,B 0,C 180,E1 -28875.754,E2 -28875.754} C_VEL
LIN {X 0,Y 72.167,Z 219.238,A -85,B 0,C 180,E1 -28878.291,E2 -28878.291} C_VEL
LIN {X 0,Y 64.656,Z 214.596,A -85,B 0,C 180,E1 -28885.967,E2 -28885.967} C_VEL
LIN {X 0,Y 59.758,Z 209.802,A -85,B 0,C 180,E1 -28896.743,E2 -28896.743} C_VEL
LIN {X 0,Y 58.178,Z 205.23,A -85,B 0,C 180,E1 -28909.08,E2 -28909.08} C_VEL
LIN {X 0,Y 58.927,Z 205.14,A -85,B 0,C 180,E1 -28918.481,E2 -28918.481} C_VEL
LIN {X 0,Y 59.194,Z 205.113,A -85,B 0,C 180,E1 -28923.787,E2 -28923.787} C_VEL
LIN {X 0,Y 58.231,Z 205.223,A -85,B 0,C 180,E1 -28936.381,E2 -28936.381} C_VEL
LIN {X 0,Y 58.163,Z 205.235,A -85,B 0,C 180,E1 -28947.74,E2 -28947.74} C_VEL
LIN {X 0,Y 58.147,Z 205.241,A -85,B 0,C 180,E1 -28951.087,E2 -28951.087} C_VEL
LIN {X 0,Y 58.515,Z 205.188,A -85,B 0,C 180,E1 -28963.873,E2 -28963.873} C_VEL
LIN {X 0,Y 58.806,Z 205.154,A -85,B 0,C 180,E1 -28973.136,E2 -28973.136} C_VEL
LIN {X 0,Y 59.381,Z 205.079,A -85,B 0,C 180,E1 -28979.999,E2 -28979.999} C_VEL
LIN {X 0,Y 58.805,Z 205.154,A -85,B 0,C 180,E1 -28986.864,E2 -28986.864} C_VEL
LIN {X 0,Y 58.515,Z 205.188,A -85,B 0,C 180,E1 -28996.126,E2 -28996.126} C_VEL
LIN {X 0,Y 58.14,Z 205.242,A -85,B 0,C 180,E1 -29008.915,E2 -29008.915} C_VEL
LIN {X 0,Y 58.149,Z 205.237,A -85,B 0,C 180,E1 -29012.239,E2 -29012.239} C_VEL
LIN {X 0,Y 58.028,Z 205.255,A -85,B 0,C 180,E1 -29017.269,E2 -29017.269} C_VEL
LIN {X 0,Y 58.012,Z 205.259,A -85,B 0,C 180,E1 -29026.625,E2 -29026.625} C_VEL
LIN {X 0,Y 58.029,Z 205.249,A -85,B 0,C 180,E1 -29032.745,E2 -29032.745} C_VEL
LIN {X 0,Y 58.152,Z 205.237,A -85,B 0,C 180,E1 -29037.777,E2 -29037.777} C_VEL
LIN {X 0,Y 58.145,Z 205.234,A -85,B 0,C 180,E1 -29041.1,E2 -29041.1} C_VEL
LIN {X 0,Y 58.523,Z 205.194,A -85,B 0,C 180,E1 -29053.886,E2 -29053.886} C_VEL
LIN {X 0,Y 58.821,Z 205.155,A -85,B 0,C 180,E1 -29063.149,E2 -29063.149} C_VEL
LIN {X 0,Y 59.394,Z 205.087,A -85,B 0,C 180,E1 -29070.011,E2 -29070.011} C_VEL
LIN {X 0,Y 58.822,Z 205.155,A -85,B 0,C 180,E1 -29076.873,E2 -29076.873} C_VEL
LIN {X 0,Y 58.654,Z 205.17,A -85,B 0,C 180,E1 -29083.876,E2 -29083.876} C_VEL
LIN {X 0,Y 58.184,Z 205.228,A -85,B 0,C 180,E1 -29091.257,E2 -29091.257} C_VEL
LIN {X 0,Y 58.132,Z 205.235,A -85,B 0,C 180,E1 -29098.932,E2 -29098.932} C_VEL
LIN {X 0,Y 58.036,Z 205.248,A -85,B 0,C 180,E1 -29107.277,E2 -29107.277} C_VEL
LIN {X 0,Y 58.139,Z 205.234,A -85,B 0,C 180,E1 -29116.509,E2 -29116.509} C_VEL
LIN {X 0,Y 58.104,Z 205.246,A -85,B 0,C 180,E1 -29122.788,E2 -29122.788} C_VEL
LIN {X 0,Y 58.009,Z 205.255,A -85,B 0,C 180,E1 -29128.022,E2 -29128.022} C_VEL
LIN {X 0,Y 57.073,Z 205.362,A -85,B 0,C 180,E1 -29135.327,E2 -29135.327} C_VEL
LIN {X 0,Y 56.715,Z 205.5,A -85,B 0,C 180,E1 -29149.606,E2 -29149.606} C_VEL
LIN {X 0,Y 57.34,Z 207.406,A -85,B 0,C 180,E1 -29154.941,E2 -29154.941} C_VEL
LIN {X 0,Y 57.977,Z 209.32,A -85,B 0,C 180,E1 -29160.472,E2 -29160.472} C_VEL
LIN {X 0,Y 60.774,Z 214.693,A -85,B 0,C 180,E1 -29176.655,E2 -29176.655} C_VEL
LIN {X 0,Y 63.568,Z 216.633,A -85,B 0,C 180,E1 -29181.019,E2 -29181.019} C_VEL
LIN {X 0,Y 64.805,Z 217.314,A -85,B 0,C 180,E1 -29182.211,E2 -29182.211} C_VEL
LIN {X 0,Y 68.047,Z 219.032,A -85,B 0,C 180,E1 -29184.402,E2 -29184.402} C_VEL
LIN {X 0,Y 69.426,Z 226.939,A -85,B 0,C 180,E1 -29187.917,E2 -29187.917} C_VEL
LIN {X 0,Y 71.738,Z 237.041,A -85,B 0,C 180,E1 -29193.76,E2 -29193.76} C_VEL
LIN {X 0,Y 75.261,Z 246.304,A -85,B 0,C 180,E1 -29199.667,E2 -29199.667} C_VEL
LIN {X 0,Y 79.782,Z 254.48,A -85,B 0,C 180,E1 -29205.182,E2 -29205.182} C_VEL
LIN {X 0,Y 78.489,Z 253.013,A -85,B 0,C 180,E1 -29207.908,E2 -29207.908} C_VEL
LIN {X 0,Y 74.229,Z 244.668,A -85,B 0,C 180,E1 -29218.445,E2 -29218.445} C_VEL
LIN {X 0,Y 73.2,Z 237.79,A -85,B 0,C 180,E1 -29226.427,E2 -29226.427} C_VEL
LIN {X 0,Y 72.476,Z 234.644,A -85,B 0,C 180,E1 -29228.305,E2 -29228.305} C_VEL
LIN {X 0,Y 71.06,Z 228.207,A -85,B 0,C 180,E1 -29231.289,E2 -29231.289} C_VEL
LIN {X 0,Y 68.336,Z 219.165,A -85,B 0,C 180,E1 -29233.393,E2 -29233.393} C_VEL
LIN {X 0,Y 60.63,Z 215.007,A -85,B 0,C 180,E1 -29239.976,E2 -29239.976} C_VEL
LIN {X 0,Y 54.625,Z 210.571,A -85,B 0,C 180,E1 -29249.988,E2 -29249.988} C_VEL
LIN {X 0,Y 51.409,Z 206.068,A -85,B 0,C 180,E1 -29263.325,E2 -29263.325} C_VEL
LIN {X 0,Y 51.312,Z 206.093,A -85,B 0,C 180,E1 -29274.247,E2 -29274.247} C_VEL
LIN {X 0,Y 52.034,Z 206.002,A -85,B 0,C 180,E1 -29282.687,E2 -29282.687} C_VEL
LIN {X 0,Y 51.876,Z 206.023,A -85,B 0,C 180,E1 -29285.622,E2 -29285.622} C_VEL
LIN {X 0,Y 51.15,Z 206.104,A -85,B 0,C 180,E1 -29296.606,E2 -29296.606} C_VEL
LIN {X 0,Y 51.055,Z 206.116,A -85,B 0,C 180,E1 -29306.59,E2 -29306.59} C_VEL
LIN {X 0,Y 51.018,Z 206.122,A -85,B 0,C 180,E1 -29315.589,E2 -29315.589} C_VEL
LIN {X 0,Y 51.456,Z 206.067,A -85,B 0,C 180,E1 -29324.146,E2 -29324.146} C_VEL
LIN {X 0,Y 51.681,Z 206.038,A -85,B 0,C 180,E1 -29332.184,E2 -29332.184} C_VEL
LIN {X 0,Y 52.265,Z 205.965,A -85,B 0,C 180,E1 -29339.999,E2 -29339.999} C_VEL
LIN {X 0,Y 51.68,Z 206.038,A -85,B 0,C 180,E1 -29347.815,E2 -29347.815} C_VEL
LIN {X 0,Y 51.382,Z 206.075,A -85,B 0,C 180,E1 -29356.82,E2 -29356.82} C_VEL
LIN {X 0,Y 51.013,Z 206.123,A -85,B 0,C 180,E1 -29364.412,E2 -29364.412} C_VEL
LIN {X 0,Y 51.022,Z 206.12,A -85,B 0,C 180,E1 -29374.286,E2 -29374.286} C_VEL
LIN {X 0,Y 50.979,Z 206.135,A -85,B 0,C 180,E1 -29386.443,E2 -29386.443} C_VEL
LIN {X 0,Y 51.045,Z 206.126,A -85,B 0,C 180,E1 -29396.598,E2 -29396.598} C_VEL
LIN {X 0,Y 51.02,Z 206.128,A -85,B 0,C 180,E1 -29405.605,E2 -29405.605} C_VEL
LIN {X 0,Y 51.464,Z 206.073,A -85,B 0,C 180,E1 -29414.163,E2 -29414.163} C_VEL
LIN {X 0,Y 51.695,Z 206.045,A -85,B 0,C 180,E1 -29422.199,E2 -29422.199} C_VEL
LIN {X 0,Y 52.279,Z 205.973,A -85,B 0,C 180,E1 -29430.012,E2 -29430.012} C_VEL
LIN {X 0,Y 51.697,Z 206.045,A -85,B 0,C 180,E1 -29437.826,E2 -29437.826} C_VEL
LIN {X 0,Y 51.378,Z 206.085,A -85,B 0,C 180,E1 -29446.76,E2 -29446.76} C_VEL
LIN {X 0,Y 51.014,Z 206.129,A -85,B 0,C 180,E1 -29454.426,E2 -29454.426} C_VEL
LIN {X 0,Y 51.018,Z 206.13,A -85,B 0,C 180,E1 -29464.257,E2 -29464.257} C_VEL
LIN {X 0,Y 51.095,Z 206.111,A -85,B 0,C 180,E1 -29476.55,E2 -29476.55} C_VEL
LIN {X 0,Y 50.943,Z 206.13,A -85,B 0,C 180,E1 -29486.507,E2 -29486.507} C_VEL
LIN {X 0,Y 50.027,Z 206.246,A -85,B 0,C 180,E1 -29495.074,E2 -29495.074} C_VEL
LIN {X 0,Y 50.374,Z 206.382,A -85,B 0,C 180,E1 -29516.001,E2 -29516.001} C_VEL
LIN {X 0,Y 55.435,Z 211.668,A -85,B 0,C 180,E1 -29530.963,E2 -29530.963} C_VEL
LIN {X 0,Y 64.805,Z 217.314,A -85,B 0,C 180,E1 -29542.211,E2 -29542.211} C_VEL
LIN {X 0,Y 66.407,Z 218.815,A -85,B 0,C 180,E1 -29544.257,E2 -29544.257} C_VEL
LIN {X 0,Y 67.185,Z 221.322,A -85,B 0,C 180,E1 -29547.089,E2 -29547.089} C_VEL
LIN {X 0,Y 67.185,Z 226.6,A -85,B 0,C 180,E1 -29552.22,E2 -29552.22} C_VEL
LIN {X 0,Y 68.243,Z 232.683,A -85,B 0,C 180,E1 -29557.104,E2 -29557.104} C_VEL
LIN {X 0,Y 70.552,Z 238.976,A -85,B 0,C 180,E1 -29561.388,E2 -29561.388} C_VEL
LIN {X 0,Y 73.693,Z 245.5,A -85,B 0,C 180,E1 -29565.666,E2 -29565.666} C_VEL
LIN {X 0,Y 74.051,Z 246.251,A -85,B 0,C 180,E1 -29567.158,E2 -29567.158} C_VEL
LIN {X 0,Y 70.141,Z 237.549,A -85,B 0,C 180,E1 -29578.165,E2 -29578.165} C_VEL
LIN {X 0,Y 69.465,Z 233.322,A -85,B 0,C 180,E1 -29583.055,E2 -29583.055} C_VEL
LIN {X 0,Y 67.664,Z 226.604,A -85,B 0,C 180,E1 -29586.257,E2 -29586.257} C_VEL
LIN {X 0,Y 65.329,Z 219.188,A -85,B 0,C 180,E1 -29587.871,E2 -29587.871} C_VEL
LIN {X 0,Y 59.167,Z 216.253,A -85,B 0,C 180,E1 -29591.855,E2 -29591.855} C_VEL
LIN {X 0,Y 52.837,Z 212.781,A -85,B 0,C 180,E1 -29598.479,E2 -29598.479} C_VEL
LIN {X 0,Y 45.766,Z 207.12,A -85,B 0,C 180,E1 -29614.39,E2 -29614.39} C_VEL
LIN {X 0,Y 45.236,Z 206.846,A -85,B 0,C 180,E1 -29616.677,E2 -29616.677} C_VEL
LIN {X 0,Y 44.458,Z 206.941,A -85,B 0,C 180,E1 -29638.293,E2 -29638.293} C_VEL
LIN {X 0,Y 44.432,Z 206.941,A -85,B 0,C 180,E1 -29649.23,E2 -29649.23} C_VEL
LIN {X 0,Y 43.924,Z 207.009,A -85,B 0,C 180,E1 -29663.108,E2 -29663.108} C_VEL
LIN {X 0,Y 43.842,Z 207.022,A -85,B 0,C 180,E1 -29671.254,E2 -29671.254} C_VEL
LIN {X 0,Y 44.221,Z 206.967,A -85,B 0,C 180,E1 -29682.421,E2 -29682.421} C_VEL
LIN {X 0,Y 44.532,Z 206.928,A -85,B 0,C 180,E1 -29690.919,E2 -29690.919} C_VEL
LIN {X 0,Y 45.14,Z 206.852,A -85,B 0,C 180,E1 -29699.999,E2 -29699.999} C_VEL
LIN {X 0,Y 44.531,Z 206.928,A -85,B 0,C 180,E1 -29709.08,E2 -29709.08} C_VEL
LIN {X 0,Y 44.145,Z 206.978,A -85,B 0,C 180,E1 -29718.566,E2 -29718.566} C_VEL
LIN {X 0,Y 43.834,Z 207.023,A -85,B 0,C 180,E1 -29728.75,E2 -29728.75} C_VEL
LIN {X 0,Y 43.797,Z 207.026,A -85,B 0,C 180,E1 -29739.931,E2 -29739.931} C_VEL
LIN {X 0,Y 43.837,Z 207.017,A -85,B 0,C 180,E1 -29753.283,E2 -29753.283} C_VEL
LIN {X 0,Y 43.838,Z 207.016,A -85,B 0,C 180,E1 -29761.269,E2 -29761.269} C_VEL
LIN {X 0,Y 44.229,Z 206.976,A -85,B 0,C 180,E1 -29772.44,E2 -29772.44} C_VEL
LIN {X 0,Y 44.544,Z 206.936,A -85,B 0,C 180,E1 -29780.937,E2 -29780.937} C_VEL
LIN {X 0,Y 45.154,Z 206.861,A -85,B 0,C 180,E1 -29790.014,E2 -29790.014} C_VEL
LIN {X 0,Y 44.545,Z 206.936,A -85,B 0,C 180,E1 -29799.092,E2 -29799.092} C_VEL
LIN {X 0,Y 44.148,Z 206.983,A -85,B 0,C 180,E1 -29808.58,E2 -29808.58} C_VEL
LIN {X 0,Y 43.824,Z 207.017,A -85,B 0,C 180,E1 -29818.774,E2 -29818.774} C_VEL
LIN {X 0,Y 43.828,Z 207.017,A -85,B 0,C 180,E1 -29829.915,E2 -29829.915} C_VEL
LIN {X 0,Y 43.84,Z 207.021,A -85,B 0,C 180,E1 -29840.116,E2 -29840.116} C_VEL
LIN {X 0,Y 43.821,Z 207.021,A -85,B 0,C 180,E1 -29843.335,E2 -29843.335} C_VEL
LIN {X 0,Y 43.243,Z 207.098,A -85,B 0,C 180,E1 -29850.82,E2 -29850.82} C_VEL
LIN {X 0,Y 42.506,Z 207.187,A -85,B 0,C 180,E1 -29860.691,E2 -29860.691} C_VEL
LIN {X 0,Y 44.714,Z 207.003,A -85,B 0,C 180,E1 -29883.38,E2 -29883.38} C_VEL
LIN {X 0,Y 52.017,Z 212.426,A -85,B 0,C 180,E1 -29898.92,E2 -29898.92} C_VEL
LIN {X 0,Y 60.797,Z 217,A -85,B 0,C 180,E1 -29907.542,E2 -29907.542} C_VEL
LIN {X 0,Y 64.938,Z 219.1,A -85,B 0,C 180,E1 -29910.261,E2 -29910.261} C_VEL
LIN {X 0,Y 66.449,Z 226.231,A -85,B 0,C 180,E1 -29913.73,E2 -29913.73} C_VEL
LIN {X 0,Y 70.094,Z 237.902,A -85,B 0,C 180,E1 -29920.697,E2 -29920.697} C_VEL
LIN {X 0,Y 70.552,Z 238.976,A -85,B 0,C 180,E1 -29921.388,E2 -29921.388} C_VEL
LIN {X 0,Y 70.836,Z 239.907,A -85,B 0,C 180,E1 -29922.687,E2 -29922.687} C_VEL
LIN {X 0,Y 70.602,Z 240,A -85,B 0,C 180,E1 -29924.756,E2 -29924.756} C_VEL
LIN {X 0,Y 69.756,Z 238.835,A -85,B 0,C 180,E1 -29927.697,E2 -29927.697} C_VEL
LIN {X 0,Y 67.689,Z 234.428,A -85,B 0,C 180,E1 -29932.946,E2 -29932.946} C_VEL
LIN {X 0,Y 66.514,Z 230.452,A -85,B 0,C 180,E1 -29937.413,E2 -29937.413} C_VEL
LIN {X 0,Y 66.175,Z 228.939,A -85,B 0,C 180,E1 -29938.897,E2 -29938.897} C_VEL
LIN {X 0,Y 64.869,Z 224.689,A -85,B 0,C 180,E1 -29940.758,E2 -29940.758} C_VEL
LIN {X 0,Y 62.909,Z 219.096,A -85,B 0,C 180,E1 -29941.886,E2 -29941.886} C_VEL
LIN {X 0,Y 53.274,Z 214.802,A -85,B 0,C 180,E1 -29947.437,E2 -29947.437} C_VEL
LIN {X 0,Y 45.188,Z 210.58,A -85,B 0,C 180,E1 -29956.495,E2 -29956.495} C_VEL
LIN {X 0,Y 40.366,Z 207.453,A -85,B 0,C 180,E1 -29966.862,E2 -29966.862} C_VEL
LIN {X 0,Y 37.027,Z 207.864,A -85,B 0,C 180,E1 -29992.291,E2 -29992.291} C_VEL
LIN {X 0,Y 37.327,Z 207.836,A -85,B 0,C 180,E1 -30004.37,E2 -30004.37} C_VEL
LIN {X 0,Y 37.173,Z 207.848,A -85,B 0,C 180,E1 -30010.863,E2 -30010.863} C_VEL
LIN {X 0,Y 36.889,Z 207.884,A -85,B 0,C 180,E1 -30019.619,E2 -30019.619} C_VEL
LIN {X 0,Y 36.772,Z 207.895,A -85,B 0,C 180,E1 -30025.013,E2 -30025.013} C_VEL
LIN {X 0,Y 37.048,Z 207.861,A -85,B 0,C 180,E1 -30041.475,E2 -30041.475} C_VEL
LIN {X 0,Y 37.326,Z 207.829,A -85,B 0,C 180,E1 -30049.146,E2 -30049.146} C_VEL
LIN {X 0,Y 37.999,Z 207.741,A -85,B 0,C 180,E1 -30059.999,E2 -30059.999} C_VEL
LIN {X 0,Y 37.325,Z 207.829,A -85,B 0,C 180,E1 -30070.852,E2 -30070.852} C_VEL
LIN {X 0,Y 37.046,Z 207.861,A -85,B 0,C 180,E1 -30078.516,E2 -30078.516} C_VEL
LIN {X 0,Y 36.714,Z 207.902,A -85,B 0,C 180,E1 -30095.048,E2 -30095.048} C_VEL
LIN {X 0,Y 36.717,Z 207.906,A -85,B 0,C 180,E1 -30100.065,E2 -30100.065} C_VEL
LIN {X 0,Y 36.719,Z 207.902,A -85,B 0,C 180,E1 -30109.96,E2 -30109.96} C_VEL
LIN {X 0,Y 36.717,Z 207.91,A -85,B 0,C 180,E1 -30114.976,E2 -30114.976} C_VEL
LIN {X 0,Y 37.054,Z 207.865,A -85,B 0,C 180,E1 -30131.503,E2 -30131.503} C_VEL
LIN {X 0,Y 37.336,Z 207.827,A -85,B 0,C 180,E1 -30139.168,E2 -30139.168} C_VEL
LIN {X 0,Y 38.013,Z 207.75,A -85,B 0,C 180,E1 -30150.017,E2 -30150.017} C_VEL
LIN {X 0,Y 37.336,Z 207.827,A -85,B 0,C 180,E1 -30160.867,E2 -30160.867} C_VEL
LIN {X 0,Y 37.054,Z 207.865,A -85,B 0,C 180,E1 -30168.498,E2 -30168.498} C_VEL
LIN {X 0,Y 36.722,Z 207.909,A -85,B 0,C 180,E1 -30185.06,E2 -30185.06} C_VEL
LIN {X 0,Y 36.747,Z 207.899,A -85,B 0,C 180,E1 -30190.093,E2 -30190.093} C_VEL
LIN {X 0,Y 36.755,Z 207.902,A -85,B 0,C 180,E1 -30199.919,E2 -30199.919} C_VEL
LIN {X 0,Y 36.537,Z 207.924,A -85,B 0,C 180,E1 -30204.757,E2 -30204.757} C_VEL
LIN {X 0,Y 35.583,Z 208.046,A -85,B 0,C 180,E1 -30216.734,E2 -30216.734} C_VEL
LIN {X 0,Y 36.577,Z 207.919,A -85,B 0,C 180,E1 -30240.001,E2 -30240.001} C_VEL
LIN {X 0,Y 40.079,Z 207.593,A -85,B 0,C 180,E1 -30252.663,E2 -30252.663} C_VEL
LIN {X 0,Y 48.156,Z 212.325,A -85,B 0,C 180,E1 -30265.966,E2 -30265.966} C_VEL
LIN {X 0,Y 57.275,Z 216.621,A -85,B 0,C 180,E1 -30273.521,E2 -30273.521} C_VEL
LIN {X 0,Y 60.666,Z 218.105,A -85,B 0,C 180,E1 -30275.398,E2 -30275.398} C_VEL
LIN {X 0,Y 62.709,Z 219.265,A -85,B 0,C 180,E1 -30276.794,E2 -30276.794} C_VEL
LIN {X 0,Y 65.447,Z 228.902,A -85,B 0,C 180,E1 -30282.157,E2 -30282.157} C_VEL
LIN {X 0,Y 69.151,Z 237.698,A -85,B 0,C 180,E1 -30287.463,E2 -30287.463} C_VEL
LIN {X 0,Y 68.699,Z 236.823,A -85,B 0,C 180,E1 -30289.44,E2 -30289.44} C_VEL
LIN {X 0,Y 66.514,Z 230.452,A -85,B 0,C 180,E1 -30297.413,E2 -30297.413} C_VEL
LIN {X 0,Y 65.77,Z 228.666,A -85,B 0,C 180,E1 -30299.061,E2 -30299.061} C_VEL
LIN {X 0,Y 63.89,Z 225.984,A -85,B 0,C 180,E1 -30300.546,E2 -30300.546} C_VEL
LIN {X 0,Y 60.629,Z 222.567,A -85,B 0,C 180,E1 -30301.555,E2 -30301.555} C_VEL
LIN {X 0,Y 57.637,Z 220.035,A -85,B 0,C 180,E1 -30301.904,E2 -30301.904} C_VEL
LIN {X 0,Y 48.69,Z 214.068,A -85,B 0,C 180,E1 -30302.834,E2 -30302.834} C_VEL
LIN {X 0,Y 44.314,Z 211.732,A -85,B 0,C 180,E1 -30305.055,E2 -30305.055} C_VEL
LIN {X 0,Y 43.513,Z 211.346,A -85,B 0,C 180,E1 -30305.797,E2 -30305.797} C_VEL
LIN {X 0,Y 36.536,Z 207.916,A -85,B 0,C 180,E1 -30316.042,E2 -30316.042} C_VEL
LIN {X 0,Y 31.871,Z 208.453,A -85,B 0,C 180,E1 -30329.98,E2 -30329.98} C_VEL
LIN {X 0,Y 29.965,Z 208.627,A -85,B 0,C 180,E1 -30350.25,E2 -30350.25} C_VEL
LIN {X 0,Y 29.91,Z 208.634,A -85,B 0,C 180,E1 -30358.006,E2 -30358.006} C_VEL
LIN {X 0,Y 29.872,Z 208.637,A -85,B 0,C 180,E1 -30375.104,E2 -30375.104} C_VEL
LIN {X 0,Y 29.515,Z 208.671,A -85,B 0,C 180,E1 -30391.559,E2 -30391.559} C_VEL
LIN {X 0,Y 29.857,Z 208.639,A -85,B 0,C 180,E1 -30400.251,E2 -30400.251} C_VEL
LIN {X 0,Y 30.1,Z 208.617,A -85,B 0,C 180,E1 -30406.496,E2 -30406.496} C_VEL
LIN {X 0,Y 30.816,Z 208.547,A -85,B 0,C 180,E1 -30419.999,E2 -30419.999} C_VEL
LIN {X 0,Y 30.099,Z 208.617,A -85,B 0,C 180,E1 -30433.502,E2 -30433.502} C_VEL
LIN {X 0,Y 29.854,Z 208.64,A -85,B 0,C 180,E1 -30439.735,E2 -30439.735} C_VEL
LIN {X 0,Y 29.486,Z 208.674,A -85,B 0,C 180,E1 -30448.469,E2 -30448.469} C_VEL
LIN {X 0,Y 29.534,Z 208.67,A -85,B 0,C 180,E1 -30465.552,E2 -30465.552} C_VEL
LIN {X 0,Y 29.491,Z 208.673,A -85,B 0,C 180,E1 -30481.56,E2 -30481.56} C_VEL
LIN {X 0,Y 29.861,Z 208.638,A -85,B 0,C 180,E1 -30490.289,E2 -30490.289} C_VEL
LIN {X 0,Y 30.109,Z 208.613,A -85,B 0,C 180,E1 -30496.523,E2 -30496.523} C_VEL
LIN {X 0,Y 30.829,Z 208.549,A -85,B 0,C 180,E1 -30510.021,E2 -30510.021} C_VEL
LIN {X 0,Y 30.109,Z 208.613,A -85,B 0,C 180,E1 -30523.52,E2 -30523.52} C_VEL
LIN {X 0,Y 29.859,Z 208.638,A -85,B 0,C 180,E1 -30529.701,E2 -30529.701} C_VEL
LIN {X 0,Y 29.492,Z 208.672,A -85,B 0,C 180,E1 -30538.488,E2 -30538.488} C_VEL
LIN {X 0,Y 29.56,Z 208.666,A -85,B 0,C 180,E1 -30555.531,E2 -30555.531} C_VEL
LIN {X 0,Y 28.756,Z 208.742,A -85,B 0,C 180,E1 -30570.739,E2 -30570.739} C_VEL
LIN {X 0,Y 28.482,Z 208.767,A -85,B 0,C 180,E1 -30590.887,E2 -30590.887} C_VEL
LIN {X 0,Y 32.008,Z 208.44,A -85,B 0,C 180,E1 -30612.685,E2 -30612.685} C_VEL
LIN {X 0,Y 36.524,Z 207.962,A -85,B 0,C 180,E1 -30623.361,E2 -30623.361} C_VEL
LIN {X 0,Y 47.669,Z 213.284,A -85,B 0,C 180,E1 -30636.139,E2 -30636.139} C_VEL
LIN {X 0,Y 58.559,Z 217.889,A -85,B 0,C 180,E1 -30642.164,E2 -30642.164} C_VEL
LIN {X 0,Y 61.415,Z 219.268,A -85,B 0,C 180,E1 -30643.929,E2 -30643.929} C_VEL
LIN {X 0,Y 64.9,Z 228.796,A -85,B 0,C 180,E1 -30649.291,E2 -30649.291} C_VEL
LIN {X 0,Y 63.98,Z 226.18,A -85,B 0,C 180,E1 -30652.82,E2 -30652.82} C_VEL
LIN {X 0,Y 63.388,Z 224.281,A -85,B 0,C 180,E1 -30654.391,E2 -30654.391} C_VEL
LIN {X 0,Y 61.454,Z 219.064,A -85,B 0,C 180,E1 -30655.405,E2 -30655.405} C_VEL
LIN {X 0,Y 50.615,Z 214.547,A -85,B 0,C 180,E1 -30660.06,E2 -30660.06} C_VEL
LIN {X 0,Y 43.513,Z 211.346,A -85,B 0,C 180,E1 -30665.797,E2 -30665.797} C_VEL
LIN {X 0,Y 38.913,Z 209.782,A -85,B 0,C 180,E1 -30670.37,E2 -30670.37} C_VEL
LIN {X 0,Y 34.083,Z 209.02,A -85,B 0,C 180,E1 -30675.569,E2 -30675.569} C_VEL
LIN {X 0,Y 25.523,Z 208.981,A -85,B 0,C 180,E1 -30691.64,E2 -30691.64} C_VEL
LIN {X 0,Y 23.14,Z 209.058,A -85,B 0,C 180,E1 -30704.463,E2 -30704.463} C_VEL
LIN {X 0,Y 22.859,Z 209.063,A -85,B 0,C 180,E1 -30709.337,E2 -30709.337} C_VEL
LIN {X 0,Y 22.504,Z 209.075,A -85,B 0,C 180,E1 -30728.616,E2 -30728.616} C_VEL
LIN {X 0,Y 22.357,Z 209.079,A -85,B 0,C 180,E1 -30741.044,E2 -30741.044} C_VEL
LIN {X 0,Y 22.809,Z 209.065,A -85,B 0,C 180,E1 -30762.052,E2 -30762.052} C_VEL
LIN {X 0,Y 23.584,Z 209.042,A -85,B 0,C 180,E1 -30779.999,E2 -30779.999} C_VEL
LIN {X 0,Y 22.802,Z 209.065,A -85,B 0,C 180,E1 -30797.95,E2 -30797.95} C_VEL
LIN {X 0,Y 22.186,Z 209.085,A -85,B 0,C 180,E1 -30819.312,E2 -30819.312} C_VEL
LIN {X 0,Y 22.187,Z 209.085,A -85,B 0,C 180,E1 -30830.728,E2 -30830.728} C_VEL
LIN {X 0,Y 22.81,Z 209.065,A -85,B 0,C 180,E1 -30852.084,E2 -30852.084} C_VEL
LIN {X 0,Y 23.595,Z 209.041,A -85,B 0,C 180,E1 -30870.027,E2 -30870.027} C_VEL
LIN {X 0,Y 22.804,Z 209.065,A -85,B 0,C 180,E1 -30887.98,E2 -30887.98} C_VEL
LIN {X 0,Y 22.203,Z 209.084,A -85,B 0,C 180,E1 -30909.312,E2 -30909.312} C_VEL
LIN {X 0,Y 21.92,Z 209.093,A -85,B 0,C 180,E1 -30920.116,E2 -30920.116} C_VEL
LIN {X 0,Y 21.143,Z 209.117,A -85,B 0,C 180,E1 -30940.587,E2 -30940.587} C_VEL
LIN {X 0,Y 29.538,Z 208.669,A -85,B 0,C 180,E1 -30988.417,E2 -30988.417} C_VEL
LIN {X 0,Y 34.324,Z 208.215,A -85,B 0,C 180,E1 -30995.515,E2 -30995.515} C_VEL
LIN {X 0,Y 48.784,Z 214.22,A -85,B 0,C 180,E1 -31006.082,E2 -31006.082} C_VEL
LIN {X 0,Y 56.043,Z 217.086,A -85,B 0,C 180,E1 -31008.801,E2 -31008.801} C_VEL
LIN {X 0,Y 54.746,Z 216.57,A -85,B 0,C 180,E1 -31010.054,E2 -31010.054} C_VEL
LIN {X 0,Y 42.715,Z 211.738,A -85,B 0,C 180,E1 -31015.354,E2 -31015.354} C_VEL
LIN {X 0,Y 34.339,Z 208.205,A -85,B 0,C 180,E1 -31023.383,E2 -31023.383} C_VEL
LIN {X 0,Y 27.978,Z 208.814,A -85,B 0,C 180,E1 -31035.428,E2 -31035.428} C_VEL
LIN {X 0,Y 22.859,Z 209.063,A -85,B 0,C 180,E1 -31069.337,E2 -31069.337} C_VEL
LIN {X 0,Y 22.096,Z 209.088,A -85,B 0,C 180,E1 -31077.164,E2 -31077.164} C_VEL
LIN {X 0,Y 20.648,Z 209.134,A -85,B 0,C 180,E1 -31084.955,E2 -31084.955} C_VEL
LIN {X 0,Y 18.576,Z 209.178,A -85,B 0,C 180,E1 -31094.899,E2 -31094.899} C_VEL
LIN {X 0,Y 15.464,Z 209.182,A -85,B 0,C 180,E1 -31122.662,E2 -31122.662} C_VEL
LIN {X 0,Y 15.689,Z 209.178,A -85,B 0,C 180,E1 -31133.286,E2 -31133.286} C_VEL
LIN {X 0,Y 16.25,Z 209.178,A -85,B 0,C 180,E1 -31139.998,E2 -31139.998} C_VEL
LIN {X 0,Y 15.247,Z 209.178,A -85,B 0,C 180,E1 -31162.908,E2 -31162.908} C_VEL
LIN {X 0,Y 15.058,Z 209.178,A -85,B 0,C 180,E1 -31167.819,E2 -31167.819} C_VEL
LIN {X 0,Y 15.063,Z 209.178,A -85,B 0,C 180,E1 -31202.237,E2 -31202.237} C_VEL
LIN {X 0,Y 15.253,Z 209.178,A -85,B 0,C 180,E1 -31207.142,E2 -31207.142} C_VEL
LIN {X 0,Y 16.258,Z 209.178,A -85,B 0,C 180,E1 -31230.039,E2 -31230.039} C_VEL
LIN {X 0,Y 15.257,Z 209.178,A -85,B 0,C 180,E1 -31252.893,E2 -31252.893} C_VEL
LIN {X 0,Y 14.839,Z 209.178,A -85,B 0,C 180,E1 -31276.703,E2 -31276.703} C_VEL
LIN {X 0,Y 14.651,Z 209.178,A -85,B 0,C 180,E1 -31320.002,E2 -31320.002} C_VEL
LIN {X 0,Y 23.315,Z 209.049,A -85,B 0,C 180,E1 -31357.078,E2 -31357.078} C_VEL
LIN {X 0,Y 30.403,Z 208.589,A -85,B 0,C 180,E1 -31366.065,E2 -31366.065} C_VEL
LIN {X 0,Y 33.168,Z 208.325,A -85,B 0,C 180,E1 -31370.507,E2 -31370.507} C_VEL
LIN {X 0,Y 23.857,Z 209.033,A -85,B 0,C 180,E1 -31382.105,E2 -31382.105} C_VEL
LIN {X 0,Y 15.481,Z 209.178,A -85,B 0,C 180,E1 -31434.772,E2 -31434.772} C_VEL
LIN {X 0,Y 15.156,Z 209.178,A -85,B 0,C 180,E1 -31472.371,E2 -31472.371} C_VEL
LIN {X 0,Y 15.689,Z 209.178,A -85,B 0,C 180,E1 -31493.286,E2 -31493.286} C_VEL
LIN {X 0,Y 15.288,Z 209.178,A -85,B 0,C 180,E1 -31499.22,E2 -31499.22} C_VEL
LIN {X 0,Y 13.095,Z 209.178,A -85,B 0,C 180,E1 -31507.736,E2 -31507.736} C_VEL
LIN {X 0,Y 7.504,Z 209.178,A -85,B 0,C 180,E1 -31538.483,E2 -31538.483} C_VEL
LIN {X 0,Y 7.32,Z 209.178,A -85,B 0,C 180,E1 -31549.772,E2 -31549.772} C_VEL
LIN {X 0,Y 7.759,Z 209.178,A -85,B 0,C 180,E1 -31564.922,E2 -31564.922} C_VEL
LIN {X 0,Y 8.684,Z 209.178,A -85,B 0,C 180,E1 -31590.073,E2 -31590.073} C_VEL
LIN {X 0,Y 7.862,Z 209.178,A -85,B 0,C 180,E1 -31616.639,E2 -31616.639} C_VEL
LIN {X 0,Y 7.241,Z 209.178,A -85,B 0,C 180,E1 -31680.004,E2 -31680.004} C_VEL
LIN {X 0,Y 15.035,Z 209.178,A -85,B 0,C 180,E1 -31726.748,E2 -31726.748} C_VEL
LIN {X 0,Y 15.84,Z 209.178,A -85,B 0,C 180,E1 -31733.709,E2 -31733.709} C_VEL
LIN {X 0,Y 9.112,Z 209.178,A -85,B 0,C 180,E1 -31769.93,E2 -31769.93} C_VEL
LIN {X 0,Y 7.892,Z 209.178,A -85,B 0,C 180,E1 -31797.047,E2 -31797.047} C_VEL
LIN {X 0,Y 7.822,Z 209.178,A -85,B 0,C 180,E1 -31833.778,E2 -31833.778} C_VEL
LIN {X 0,Y 8.677,Z 209.178,A -85,B 0,C 180,E1 -31859.996,E2 -31859.996} C_VEL
LIN {X 0,Y 7.754,Z 209.178,A -85,B 0,C 180,E1 -31885.18,E2 -31885.18} C_VEL
LIN {X 0,Y 7.32,Z 209.178,A -85,B 0,C 180,E1 -31909.772,E2 -31909.772} C_VEL
LIN {X 0,Y 7.747,Z 211.178,A -85,B 0,C 180,E1 -31924.68,E2 -31924.68} C_VEL
LIN {X 0,Y 7.747,Z 600,A -85,B 0,C 180,E1 -31924.68,E2 -31924.68} C_VEL
LIN {X 0,Y 7.747,Z 600,A -85,B 0,C 180,E1 -31924.68,E2 -31924.68}

QRS_NEXT_CUT()

QRS_NEXT()
QRS_HOME()

END
